// oscat_building/POUs/Jalousie/BLIND_CONTROL
FUNCTION_BLOCK BLIND_CONTROL
VAR_INPUT
	UP, DN : BOOL;
	S_IN : BYTE;
	PI : BYTE;
	AI : BYTE;
	T_UD, T_ANGLE : TIME;
END_VAR
VAR_INPUT CONSTANT
	SENS : BYTE := 5;
	T_LOCKOUT: TIME := T#100ms;
END_VAR
VAR_OUTPUT
	POS, ANG : BYTE;
	MU, MD : BOOL;
	STATUS : BYTE;
END_VAR
VAR
	act : BLIND_ACTUATOR;
	delta : BYTE;
	bTimeTest:BOOL:=FALSE;
	iPos:BYTE;
	iAngel:BYTE;
END_VAR

(*
version 1.5		8. mar 2011
programmer 		AE
tested by		AE

*)

IF bTimeTest THEN
	PI:=iPos;
	AI:=iAngel;
	UP:=TRUE;
	DN:=TRUE;
END_IF

(* Check Position*)
act(T_UD:=T_UD, T_ANGLE:=T_ANGLE, T_lockout := T_Lockout);

IF UP AND DN THEN
	(* automatic modus detected *)
	(* first find correct position *)
	IF BYTE_TO_INT(act.pos) < BYTE_TO_INT(pi) - delta THEN
		act.UP := TRUE;
		act.DN := FALSE;
		delta := 0;
		STATUS := 121;
	ELSIF BYTE_TO_INT(act.pos) > BYTE_TO_INT(pi) + delta THEN
		act.UP := FALSE;
		act.DN := TRUE;
		delta := 0;
		STATUS := 122;
	(* regulate angle *)
	ELSIF BYTE_TO_INT(act.ang) < BYTE_TO_INT(ai) - delta AND T_angle > T#100ms THEN
		act.UP := TRUE;
		act.DN := FALSE;
		delta := sens/2;
		STATUS := 123;
	ELSIF BYTE_TO_INT(act.ang) > BYTE_TO_INT(ai) + delta AND T_angle > T#100ms THEN
		act.UP := FALSE;
		act.DN := TRUE;
		delta := sens/2;
		STATUS := 124;
	(* correct position reached *)
	ELSE
		act.UP := FALSE;
		act.DN := FALSE;
		delta := sens;
		STATUS := S_IN;
	END_IF;
ELSE
	act.UP := UP;
	act.DN := DN;
	STATUS := S_IN;
END_IF;

(* blind control calls blind_actuator *)
act(T_UD:=T_UD, T_ANGLE:=T_ANGLE, T_lockout := T_Lockout);
pos := act.pos;
ang := act.ang;
MU := act.QU;
md := act.QD;
status := act.status;

(* revision history
hm	29. sep 2007	rev 1.0
	original release

hm	6. oct 2007	rev 1.1
	rearranged outputs
	integrated blind_actuator into blind_control

hm	16. oct 2007	rev 1.2
	ignore angle when t_angle = 0

hm 29. oct 2007	rev 1.3
	added lockout configuration time for motor direction change
	sens has a setup value of 5

hm	27. jul. 2009	rev 1.4
	changed status handling

ae	08. mar. 2010	rev 1.5
	at aPosition bevor control
	at tolerance "delta := sens/2;"

*)

END_FUNCTION_BLOCK

// oscat_building/POUs/Jalousie/BLIND_CONTROL_S
FUNCTION_BLOCK BLIND_CONTROL_S
VAR_INPUT
	UP, DN : BOOL;
	S_IN : BYTE := 125;
	PI : BYTE;
	T_UP : TIME;
	T_DN : TIME;
	RU : BOOL;
	RD : BOOL;
END_VAR
VAR_INPUT CONSTANT
	T_LOCKOUT: TIME := T#100ms;
	T_EXT : TIME;
	EXT_TRIG : BYTE := 5;
	R_POS_TOP : BYTE := 255;
	R_POS_BOT : BYTE;
END_VAR
VAR_OUTPUT
	POS : BYTE;
	MU, MD : BOOL;
	STATUS : BYTE;
END_VAR
VAR
	rmp : _RMP_NEXT;
	tx, last : TIME;
	PI_last: BYTE;
END_VAR


(*
version 1.2	23. jan 2010
programmer 	hugo
tested by		heinz


*)


(* status definition
	121 = manual up				manual up operation UP = true and DN = false
	122 = manual down			manual down operation DN = true and UP = false
	123 = auto positioning		automatic mode DN = UP = TRUE
	124 = revert					revert from top or bottom
	125 = nothing					default input for S_IN
	127 = Lockout time			lockout between directional change
	128 = calibrate				calibrate after power up
	129 = extend					extend runtime at top or bottom for continuous calibration
*)

(* read system time *)
tx := DWORD_TO_TIME(T_PLC_MS());

(* check inputs and start state machine *)
IF UP  AND NOT DN THEN
	(*  manual UP *)
	rmp.IN := 255;
	STATUS := 121;
ELSIF DN AND NOT UP THEN
	(* manual DN *)
	rmp.IN := 0;
	STATUS := 122;
ELSIF NOT (UP OR DN) THEN
	(* manual standby mode *)
	rmp.IN := PI;
	STATUS := S_IN;
END_IF;

(* simulate pos output *)
rmp(E := UP OR DN, TR := T_UP, TF := T_DN, TL := T_LOCKOUT, OUT := POS);

(* state machine *)
CASE STATUS OF
	0:		(* power up init *)
		last := tx;
		PI_last := PI XOR BYTE#255;
		STATUS := 128;		(* calibrate *)

	121: 	(* manual up *)
		MU := TRUE;
		MD := FALSE;
		IF POS >= (BYTE#255 - EXT_TRIG) THEN
			(* extend cycle if top is reached *)
			POS := 255;
			last := tx;
			STATUS := 129;	(* extend *)
		END_IF;

	122:	(* manual down *)
		MD := TRUE;
		MU := FALSE;
		IF POS <= EXT_TRIG THEN
			(* extend cycle if bottom is reached *)
			POS := 0;
			last := tx;
			STATUS := 129;	(* extend *)
		END_IF;

	123:	(* auto positioning *)
		MD := rmp.DN;
		MU := rmp.UP;
		IF NOT (rmp.DN OR rmp.UP) THEN
			(* automatic position is reached *)
			IF POS <= EXT_TRIG THEN
				(* extend at bottom *)
				MD := TRUE;
				last := tx;
				STATUS := 129;	(* extend *)
			ELSIF POS >= (BYTE#255 - EXT_TRIG)  THEN
				(* extend at top *)
				MU := TRUE;
				last := tx;
				STATUS := 129;	(* extend *)
			ELSE
				STATUS := S_IN;
			END_IF;
		END_IF;

	124:	(* revert from top or bottom *)
		MD := rmp.DN;
		MU := rmp.UP;
		IF NOT(rmp.DN OR rmp.UP) THEN
(*		IF POS = rmp.IN THEN  *)
			PI_last := PI;
			STATUS := S_IN;
		END_IF;

	127:	(* lockout time *)
		IF (tx - last) >= T_LOCKOUT THEN
				STATUS := S_IN;
		END_IF;

	128:	(* calibration *)
		MU := TRUE;
		MD := FALSE;
		rmp.IN := 255;
		IF (tx - last) >= (T_UP +  T_EXT) THEN
			MU := FALSE;
			last := tx;
			STATUS := 127;	(* lockout *)
		END_IF;

	129: (* extend mode *)
		IF (tx - last) >= T_EXT THEN
			MU := FALSE;
			MD := FALSE;
			last := tx;
			STATUS := 127;	(* lockout *)
		END_IF;

ELSE
	MU := FALSE;
	MD := FALSE;
	IF PI <> PI_last THEN
		PI_last := PI;
		rmp.IN := PI;
		STATUS := 123;	(* auto positioning *)
	ELSIF POS = 0 AND RU THEN
		rmp.IN := R_POS_BOT;
		STATUS := 124;	(* revert *)
	ELSIF pos = 255 AND RD THEN
		rmp.IN := R_POS_TOP;
		STATUS := 124;	(* revert *)
	ELSE
		STATUS := S_IN;
	END_IF;
END_CASE;



(* revision history

hm	9. mar. 2009	rev 1.0
	original release

hf	27. jul 2009	rev 1.1
	major code changes and updates

hf	23. Jan 2010	rev 1.2
	fixed a bug during calibration
	added T_UP and T_DN

*)

END_FUNCTION_BLOCK

// oscat_building/POUs/Jalousie/BLIND_INPUT
FUNCTION_BLOCK BLIND_INPUT
VAR_INPUT
	POS, ANG : BYTE;
	S1, S2 : BOOL;
	IN : BOOL;
	PI, AI : BYTE;
END_VAR
VAR_INPUT CONSTANT
	SINGLE_SWITCH : BOOL;
	CLICK_EN : BOOL := TRUE;
	CLICK_TIME : TIME := T#500ms;
	MAX_RUNTIME : TIME := T#60s;
	MANUAL_TIMEOUT: TIME := T#1h;
	DEBOUNCE_TIME : TIME := T#20ms;
	DBL_CLK1 : BOOL := FALSE;
	DBL_POS1 : BYTE;
	DBL_ANG1 : BYTE;
	DBL_CLK2 : BOOL := FALSE;
	DBL_POS2 : BYTE := 255;
	DBL_ANG2 : BYTE := 255;
	D1_TOGGLE : BOOL := TRUE;
	D2_TOGGLE : BOOL := TRUE;
	MASTER_MODE : BOOL;
END_VAR
VAR_OUTPUT
	QU : BOOL := TRUE;
	QD : BOOL := TRUE;
	STATUS : BYTE;
	PO : BYTE := 255;
	AO : BYTE := 255;
	D1, D2 : BOOL;
END_VAR
VAR
	s1e, s2e : TOF;
	s1d, s2d : CLICK_MODE;
	dir : BOOL;
	tx, last : TIME;
END_VAR

(*
version 1.7	12. nov. 2009
programmer 	hugo
tested by		oscat


*)

(* read system timer *)
tx := DWORD_TO_TIME(T_PLC_MS());

(* inputs S1 and S2 are debounced and then decoded for multiple clicks *)
s1e(in := S1, pt := DEBOUNCE_TIME);
s2e(in := S2, pt := DEBOUNCE_TIME);
s1d(in := (s1e.Q AND NOT SINGLE_SWITCH) OR (s1e.Q AND SINGLE_SWITCH AND dir), t_long := CLICK_TIME);
s2d(in := (s2e.Q AND NOT SINGLE_SWITCH) OR (s1e.Q AND SINGLE_SWITCH AND NOT dir), t_long := CLICK_TIME);

(* if d1 and d2 are not toggle clear them to make sure they are only active for oine cycle *)
IF NOT d1_toggle THEN d1 := FALSE; END_IF;
IF NOT d2_toggle THEN d2 := FALSE; END_IF;

(* decode actions *)
IF (s1d.LONG AND s2d.LONG) OR (status = 139) THEN
   status := 139;
   IF NOT (s1d.LONG OR s2d.LONG)  THEN status := 130; END_IF;
ELSIF s1d.tp_LONG THEN
	status := 132;
ELSIF s2d.tp_LONG THEN
	status := 133;
ELSIF  s1d.SINGLE THEN
	IF click_en THEN
		(* if running then we stop otherwise start new direction *)
		IF QU XOR QD THEN
			status := 131;
		ELSE
			status := 134;
			last := tx;
			dir := NOT dir;
		END_IF;
	END_IF;
ELSIF  s2d.SINGLE THEN
	IF click_en THEN
		(* if running then we stop otherwise start new direction *)
		IF QU XOR QD THEN
			status := 131;
		ELSE
			status := 135;
			last := tx;
			dir := NOT dir;
		END_IF;
	END_IF;
ELSIF in THEN
	status := 136;
	last := tx;
ELSIF s1d.DOUBLE THEN
	IF dbl_clk1 THEN
		(* a position need to be set for a double click on S1 *)
		status := 137;
		last := tx;
	ELSE
		(* toggle the output when dbl_clk1 is not active *)
		D1 := NOT D1;
	END_IF;
ELSIF s2d.DOUBLE THEN
	IF dbl_clk2 THEN
		(* a position need to be set for a double click on S2 *)
		status := 138;
		last := tx;
	ELSE
		(* toggle the output when dbl_clk2 is not active *)
		(* in single switch mode we need to toggle d1 instead of d2 *)
		IF single_switch THEN D1 := NOT D1; ELSE D2 := NOT D2; END_IF;
	END_IF;
END_IF;


(* state machine *)
CASE status OF
	0:		(* power up operation *)
			status := 130;

	130:	(* automatic operation standby *)
			IF NOT master_mode THEN
				PO := POS;
				AO := ANG;
			END_IF;
			QU := TRUE;
			QD := TRUE;

	131:	(* manual operation standby *)
			QU := FALSE;
			QD := FALSE;
			PO := POS;
			AO := ANG;
			(* manual mode will be ended when timeout is reached *)
			IF tx - last >= manual_timeout THEN
				status := 130;
			END_IF;

	132:	(* manual operation up *)
			QU := TRUE;
			QD := FALSE;
			PO := POS; AO := ANG;
			last := tx;
			IF NOT s1d.LONG THEN status := 131; dir := NOT dir; END_IF;

	133:	(* manual operation down *)
			QU := FALSE;
			QD := TRUE;
			PO := POS; AO := ANG;
			last := tx;
			IF NOT s2d.LONG THEN	status := 131; dir := NOT dir; END_IF;

	134:	(* manual operation single click up *)
			QU := TRUE;
			QD := FALSE;
			PO := POS; AO := ANG;
			IF tx - last >= max_runtime THEN status := 131; END_IF;

	135:	(* manual operation single click dn *)
			QU := FALSE;
			QD := TRUE;
			PO := POS; AO := ANG;
			IF tx - last >= max_runtime THEN status := 131;	END_IF;

	136:	(* forced input in = true *)
			QU := TRUE;
			QD := TRUE;
			PO := PI; AO := AI;
			IF tx-last >= max_runtime THEN status := 130; END_IF;

	137:	(* double click1 position *)
			QU := TRUE;
			QD := TRUE;
			PO := DBL_POS1;
			AO := DBL_ANG1;
			IF tx - last >= max_runtime THEN status := 131; END_IF;

	138:	(* double click2 position *)
			QU := TRUE;
			QD := TRUE;
			PO := DBL_POS2;
			AO := DBL_ANG2;
			IF tx - last >= max_runtime THEN status := 131; END_IF;

	   139:   (* manual operation standby *)
	         QU := FALSE;
	         QD := FALSE;
	         PO := POS;
	         AO := ANG;

END_CASE;


(* revision history
hm	29. sep 2007	rev 1.0
	original release

hm	6. oct 2007		rev 1.1
	renamed ps and as to po and ao

hm	30. dec 2007	rev 1.2
	added click_timeout variable and function

hm	16. jul. 2008	rev 1.3
	rewirtten code to allow for more functionality
	added single click mode with single_switch.
	added Debounce for inputs S1 and S2
	added double_click functionality

hm	26. sep. 2008	rev 1.4
	corrected an error while POS and ANG was transferred to outputs PO and AO during automatic modes

hm	22. jan 2009	rev 1.5
	added pulse mode for double click outputs
	added automatic mode for IN

hm	27. jul 2009	rev 1.6
	changed status 0 to 130

HF	12. nov. 2009	rev 1.7
	added state 139
	set defaults for QU, QD, PO

*)

END_FUNCTION_BLOCK

// oscat_building/POUs/Jalousie/BLIND_NIGHT
FUNCTION_BLOCK BLIND_NIGHT
VAR_INPUT
	UP, DN : BOOL;
	S_IN : BYTE;
	PI, AI : BYTE;
	E_NIGHT : BOOL := TRUE;
	E_DAY	: BOOL := TRUE;
	DTIN : DT;
	SUNRISE, SUNSET : TOD;
END_VAR
VAR_INPUT CONSTANT
	SUNRISE_OFFSET : TIME;
	SUNSET_OFFSET : TIME;
	NIGHT_POSITION : BYTE;
	NIGHT_ANGLE : BYTE;
END_VAR
VAR_OUTPUT
	QU, QD : BOOL;
	STATUS : BYTE;
	PO, AO : BYTE;
END_VAR
VAR
	night : BOOL;
	last_night, last_day : DATE;
END_VAR

(*
version 1.2	6 oct 2007
programmer 	hugo
tested by		tobias


*)

IF NOT (up AND dn) AND night THEN
	(* manual operation at night will cancel operation for one night *)
	night := FALSE;
ELSIF (DT_TO_TOD(dtin) > sunset + sunset_offset) AND (last_night < DT_TO_DATE(dtin)) AND NOT night AND e_night THEN
	(* enable night *)
	night := TRUE;
	last_night := DT_TO_DATE(dtin);
ELSIF (DT_TO_TOD(dtin) > sunrise + sunrise_offset) AND (last_day < DT_TO_DATE(dtin)) AND night AND e_day AND (last_night < DT_TO_DATE(dtin)) THEN
	(* disable night *)
	night := FALSE;
	last_day := DT_TO_DATE(dtin);
END_IF;

(* shade at night only in auto mode and enable = true *)
IF UP AND DN AND night THEN
	status := 141;
	po := night_position;
	ao := night_angle;
ELSE
	QU := UP;
	QD := DN;
	po := pi;
	ao := ai;
	status := s_in;
END_IF;


(* revision history
hm	29. sep 2007	rev 1.0
	original version

hm	5. oct 2007		rev 1.1
	added enable input

hm	6. oct 2007		rev 1.2
	added pos and angle inputs and outputs
	night position and angle can now be configured
	any manual operation at night will cancel night operation

*)

END_FUNCTION_BLOCK

// oscat_building/POUs/Jalousie/BLIND_SCENE
FUNCTION_BLOCK BLIND_SCENE
VAR_INPUT
	UP, DN : BOOL;
	S_IN : BYTE;
	PI, AI : BYTE;
	ENABLE : BOOL;
	SWRITE : BOOL;
	SCENE : BYTE;
END_VAR
VAR_OUTPUT
	QU, QD : BOOL;
	STATUS : BYTE;
	PO, AO : BYTE;
END_VAR
VAR RETAIN
	sx : ARRAY[0..15,0..2] OF BYTE;
END_VAR
VAR_TEMP
	x : BYTE;
END_VAR

(*
version 1.1	29. jan 2008
programmer 	hugo
tested by		tobias


*)

(* delete all bits except the lower 4 of scene *)
x := scene AND 16#0F;

IF enable AND sx[x,2] > 0 AND UP AND DN THEN
	po := sx[x,0];
	ao := sx[x,1];
	status := 160 + x;  (* Status number is 160 to 175 for the 16 scenes *)
	QU := TRUE;
	QD := TRUE;
ELSE
	QU := UP;
	QD := DN;
	status := S_IN;
	po := pi;
	ao := ai;
END_IF;

(* write scene if necessary *)
IF swrite THEN
	status := 176;		(* write scene *)
	sx[x,0] := pi;
	sx[x,1] := ai;
	IF enable THEN sx[x,2] := 1; ELSE sx[x,2] := 0; END_IF; (* if sx[x,2] = 0 the scene is disabled *)
END_IF;


(* revision history
hm	24. oct 2007	rev 1.0
	original release

hm		29.1.2008	rev 1.1
	replaced shr/shl with and for better performance
*)

END_FUNCTION_BLOCK

// oscat_building/POUs/Jalousie/BLIND_SECURITY
FUNCTION_BLOCK BLIND_SECURITY
VAR_INPUT
	UP, DN : BOOL;
	S_IN : BYTE;
	PI, AI : BYTE;
	FIRE : BOOL;
	WIND : BOOL;
	ALARM : BOOL;
	DOOR : BOOL;
	RAIN : BOOL;
END_VAR
VAR_INPUT CONSTANT
	Alarm_UP : BOOL := TRUE;
	WIND_UP :BOOL := TRUE;
	RAIN_UP : BOOL := FALSE;
END_VAR
VAR_OUTPUT
	QU, QD : BOOL;
	STATUS : BYTE;
	PO, AO : BYTE;
END_VAR


(*
version 1.2	12. feb 2008
programmer 	hugo
tested by		tobias


*)

IF Fire THEN
	QU := TRUE;
	QD := FALSE;
	status := 111;
ELSIF Wind THEN
	QU := Wind_up;
	QD := NOT wind_up;
	status := 112;
ELSIF alarm THEN
	QU := Alarm_up;
	QD := NOT Alarm_up;
	status := 113;
ELSIF Door THEN
	QU := TRUE;
	QD := FALSE;
	status := 114;
ELSIF Rain AND NOT (up XOR dn) THEN
	QU := rain_up;
	QD := NOT rain_up;
	status := 115;
ELSE
	QU := UP;
	QD := DN;
	status := S_IN;
	po := pi;
	ao := ai;
END_IF;


(* revision history
hm	29. sep 2007	rev 1.0
	original release

hm	6. oct 2007		rev 1.1
	added pos and angle inputs and outputs
	manual will override rain position
	alarm position can now be configured

hm		12. feb. 2008	rev 1.2
	added config variables rain_up and wind_up
	position for rain and wind is now configurable
*)

END_FUNCTION_BLOCK

// oscat_building/POUs/Jalousie/BLIND_SET
FUNCTION_BLOCK BLIND_SET
VAR_INPUT
	UP, DN : BOOL;
	S_IN : BYTE;
	PI, AI : BYTE;
	IN : BOOL;
	PX, AX : BYTE;
END_VAR
VAR_INPUT CONSTANT
	OVERRIDE_MANUAL : BOOL;
	RESTORE_POSITION : BOOL;
	RESTORE_TIME : TIME := T#60s;
END_VAR
VAR_OUTPUT
	QU, QD : BOOL;
	STATUS : BYTE;
	PO, AO : BYTE;
END_VAR
VAR
	tx: TIME;
	ps: BYTE;
	as: BYTE;
	last: TIME;
END_VAR

(*
version 1.0	27. jul 2009
programmer 	hugo
tested by		oscat

BLIND_SET can be used to force a definite position and angle.
blind_set can be placed close to blind_control for high priority while blind_input must be always at the beginning of the chain with low priority.

*)

(* read system time *)
tx := DWORD_TO_TIME(T_PLC_MS());

(* check inputs *)
IF IN THEN
	IF override_manual OR (UP AND DN) THEN
		status := 178;
	END_IF;
END_IF;

(* state machine *)
CASE STATUS OF
	0: (* power on state *)
		status := S_IN;

	178: (* force values from PX and AX *)
		PO := PX;
		AO := AX;
		QU := TRUE;
		QD := TRUE;
		(* check for end of forced position *)
		IF NOT in THEN
			STATUS := SEL(RESTORE_POSITION, S_IN, 179);
			last := tx;
		END_IF;

	179: (* restore previous position *)
		PO := ps;
		AO := as;
		IF ((PO = PI) AND (AO = AI))  OR tx - last >= RESTORE_TIME THEN
			status := S_IN;
		END_IF;

ELSE
	(* no operation transfer inputs to outputs *)
	PO := PI;
	ps := PI;
	AO := AI;
	as := AI;
	STATUS := S_IN;
	QU := UP;
	QD := DN;
END_CASE;


(* revision history
hm	27. jul 2009	rev 1.0
	original release

*)

END_FUNCTION_BLOCK

// oscat_building/POUs/Jalousie/BLIND_SHADE
FUNCTION_BLOCK BLIND_SHADE
VAR_INPUT
	UP, DN : BOOL;
	S_IN : BYTE;
	PI, AI : BYTE;
	ENABLE : BOOL;
	SUN : BOOL;
END_VAR
VAR_IN_OUT
	CX : CALENDAR;
END_VAR
VAR_INPUT CONSTANT
	sunrise_offset : TIME := T#1h;
	sunset_preset : TIME := T#1h;
	direction : REAL := 180.0;
	angle_offset : REAL := 80.0;
	slat_width : REAL := 80.0;
	Slat_spacing : REAL := 60.0;
	Shade_delay : TIME := T#60s;
	Shade_pos : BYTE;
END_VAR
VAR_OUTPUT
	QU, QD : BOOL;
	STATUS : BYTE;
	PO, AO : BYTE;
END_VAR
VAR
	angle: REAL;
	sun_delay : TOF;
END_VAR

(*
version 1.4	13. mar. 2009
programmer 	hugo
tested by		tobias


*)

(* the input sun is sent through tof which will delay the shade for the time shade_delay *)
sun_delay(IN := sun, PT := shade_delay);

IF UP AND DN AND enable AND sun_delay.Q AND cx.SUN_HOR > direction - angle_offset AND cx.SUN_HOR < direction + angle_offset AND
	DT_TO_TOD(cx.UTC) > cx.SUN_RISE + sunrise_offset AND DT_TO_TOD(cx.UTC) < cx.SUN_SET - sunset_preset THEN
	status := 151;
	QU := UP;
	QD := DN;
	(* position is predefined *)
	po := shade_pos;
	(* shading is active now calculate the slat angle *)
	(* calculate the max angle for the blind *)
	angle := DEG(ATAN(slat_spacing / slat_width));
	(* check if sun angle is between 0 and max angle *)
	IF cx.SUN_VER > 0.0 AND cx.SUN_VER < angle THEN
		angle := cx.SUN_VER + DEG(ACOS(COS(RAD(cx.SUN_VER))*slat_spacing / Slat_width));
		ao := DINT_TO_BYTE(LIMIT(0,TRUNC(angle * 2.833333333), 255));
	ELSE
		ao := 255;
	END_IF;
ELSE
	QU := UP;
	QD := DN;
	po := pi;
	ao := ai;
	status := S_IN;
END_IF;

(* revision history
hm	15 oct. 2007	rev 1.0
	original version

hm	19. oct 2007	rev 1.1
	manual mode was not detected because outputs were checked and not inputs UP and DN

hm	24. nov 2007	rev 1.2
	added shade_delay to avoid constant up and down if sun is out parcially

hm	8. feb 2009	rev 1.3
	added shading position shade_pos to be configured
	changed inputs to utilize calendar data structure

hm	13. mar. 2009	rev 1.4
	improved code

*)

END_FUNCTION_BLOCK

// oscat_building/POUs/Jalousie/BLIND_SHADE_S
FUNCTION_BLOCK BLIND_SHADE_S
VAR_INPUT
   UP, DN : BOOL;
   S_IN : BYTE;
   PI : BYTE;
   ENABLE : BOOL;
   SUN : BOOL;
   HORZ1 : REAL := 100.0;
   HORZ2 : REAL := 260.0;
   VERT : REAL := 90.0;
   ALERT: BOOL := FALSE;
END_VAR
VAR_IN_OUT
   CX : calendar;
END_VAR
VAR_INPUT CONSTANT
   sunrise_offset : TIME := T#1h;
   sunset_preset : TIME := T#1h;
   shade_delay : TIME := T#60s;
   shade_pos : BYTE;
END_VAR
VAR_OUTPUT
   QU, QD : BOOL;
   STATUS : BYTE;
   PO : BYTE;
END_VAR
VAR
   sun_delay : TOF;
END_VAR
(*
version 1.0	12. nov. 2009
programmer 	heinz
tested by		oscat


*)

(* status definition
   151 = shadow               move shutter down for shadowing
   152 = alert                  move shutter up by setting QU:=TRUE when door is open.
*)

(* the input sun is sent through tof which will delay the shade for the time shade_delay *)
sun_delay(IN := sun, PT := shade_delay);

IF ALERT THEN
   QU := TRUE;
   QD := FALSE;
   STATUS := 152;
ELSIF UP AND DN AND ENABLE AND sun_delay.Q
AND (CX.SUN_HOR > HORZ1) AND (CX.SUN_HOR < HORZ2)
AND (CX.SUN_VER < VERT)
AND (DT_TO_TOD(CX.UTC) > CX.SUN_RISE + sunrise_offset) AND (DT_TO_TOD(CX.UTC) < CX.SUN_SET - sunset_preset) THEN
   QU := UP;
   QD := DN;
   STATUS := 151;
   (* Calculate Position, must be shade_pos or less *)
   PO := MIN(PI, shade_pos);
ELSE
   QU := UP;
   QD := DN;
   PO := PI;
   STATUS := S_IN;
END_IF;



(* revision history
hf	12 nov. 2009	rev 1.0
	original version

*)

END_FUNCTION_BLOCK

// oscat_building/POUs/Other/BUILDING_VERSION
FUNCTION BUILDING_VERSION : DWORD
VAR_INPUT
	IN : BOOL;
END_VAR


(*
version 1.1	16 dec 2007
programmer 	hugo
tested by		oscat

oscat_version returns the version number in dword format
132 is library version 1.32
if IN = true, the release date will be returned

*)

IF in THEN
	BUILDING_VERSION := DATE_TO_DWORD(D#2011-02-3);
ELSE
	BUILDING_VERSION := 100;
END_IF;

(* revision history
hm	6. oct 2006	rev 1.0
	original version

hm	16. dec 2007	rev 1.1
	added possibility to return date and version depending on IN.

*)

END_FUNCTION

// oscat_network/POUs/CO_NVERT/BASE64_DECODE_STR_1
FUNCTION_BLOCK BASE64_DECODE_STR_1
VAR_INPUT
	RUN : BOOL;
END_VAR
VAR_OUTPUT
	DONE : BOOL;
END_VAR
VAR_IN_OUT
	STR1 : STRING(192);
	STR2 : STRING(144);
END_VAR
VAR
	BASE64_DECODE_STREAM : BASE64_DECODE_STREAM;
	run_last : BOOL;
	buf1 : ARRAY [0..63] OF BYTE;
	buf2 : ARRAY [0..47] OF BYTE;
	mode : INT;
	size1 : INT;
	size2 : INT;
	end : INT;
	pos : INT;
END_VAR

(*
version 1.0	06. dec. 2009
programmer 	ks
tested by	ks

BASE64_DECODE_STR konvertiert einen BASE64 kodierten String in einen normalen String. 

*)

CASE mode OF
0:	IF RUN AND NOT run_last THEN
		DONE := FALSE;
		mode := 1;
		end := LEN(STR1);
		pos := 0;
		STR2 := '';
	END_IF;
1:
	size1 := MIN(48,end - pos);
	IF size1 > 0 THEN
		_STRING_TO_BUFFER(STR:=MID(STR1, size1, pos + 1), POS:=0, PT:=ADR(buf1), SIZE:=SIZEOF(buf1));
		BASE64_DECODE_STREAM(BUF1:=buf1 ,BUF2:=buf2 ,SIZE1:=size1 ,SIZE2=>size2);
		STR2 := CONCAT(STR2,BUFFER_TO_STRING(PT:=ADR(buf2), SIZE:=SIZEOF(buf2), START:=0, STOP:=size2 - 1));
	ELSE
		mode := 0;
		DONE := TRUE;
	END_IF;
	pos := pos + size1;
END_CASE;

run_last := RUN;

(* revision history

ks	6. dec. 2009 rev 1.0
	original version

*)

END_FUNCTION_BLOCK

// oscat_network/POUs/CO_NVERT/BASE64_DECODE_STREAM_1
FUNCTION_BLOCK BASE64_DECODE_STREAM_1
VAR_IN_OUT
	BUF1 : ARRAY [0..63] OF BYTE;
	BUF2 : ARRAY [0..47] OF BYTE;
END_VAR
VAR_INPUT
	SIZE1 : INT;
END_VAR
VAR_OUTPUT
	SIZE2 : INT;
END_VAR
VAR_TEMP
	a: INT;
	b: WORD;
	o: INT;
	off: INT;
	i1: INT;
	i2: INT;
	c: INT;
END_VAR

(*
version 1.0	06. dec. 2009
programmer 	ks
tested by	ks

BASE64_DECODE_STREAM konvertiert einzelne Base64 kodierte Datenblöcke in normalen Datenblöcke. 

*)

IF SIZE1 <= 0 THEN SIZE2 := 0; RETURN; END_IF;
c := SIZE1 - 1;
i2 := 0;
a := 0;
b := 0;
FOR i1 := 0 TO c DO
	o := BUF1[i1];
	IF o = 61  (* = *) THEN	EXIT;
	ELSIF o > 96 (* a-z *) THEN off := 71;
	ELSIF o > 64 (* A-Z *) THEN off := 65;
	ELSIF o > 47 (* 0-9 *) THEN off := -4;
	ELSIF o = 43 (* + *) THEN off := -19;
	ELSIF o = 47 (* / *) THEN off := -16;
	END_IF;
	b := SHL(b,6) OR INT_TO_BYTE(o - off);
	a := a + 6;
	IF a >= 8 THEN
		a := a - 8;
		BUF2[i2] := WORD_TO_BYTE(SHR(b,a));
		i2 := i2 + 1;
		b := b AND NOT SHL(WORD#16#FFFF,a);
	END_IF;
END_FOR;
SIZE2 := i2;

(* revision history

ks	6. dec. 2009 rev 1.0
	original version

*)

END_FUNCTION_BLOCK

// oscat_network/POUs/CO_NVERT/BASE64_ENCODE_STR_1
FUNCTION_BLOCK BASE64_ENCODE_STR_1
VAR_INPUT
	RUN : BOOL;
END_VAR
VAR_OUTPUT
	DONE : BOOL;
END_VAR
VAR_IN_OUT
	STR1 : STRING(144);
	STR2 : STRING(192);
END_VAR
VAR
	BASE64_ENCODE_STREAM : BASE64_ENCODE_STREAM;
	run_last : BOOL;
	buf1 : ARRAY [0..47] OF BYTE;
	buf2 : ARRAY [0..63] OF BYTE;
	mode : INT;
	size1 : INT;
	size2 : INT;
	end : INT;
	pos : INT;
END_VAR

(*
version 1.0	06. dec. 2009
programmer 	ks
tested by	ks

BASE64_ENCODE_STR konvertiert einen normalen String in einen BASE64 kodierten String. 

*)

CASE mode OF
0:	IF RUN AND NOT run_last THEN
		DONE := FALSE;
		mode := 1;
		end := LEN(STR1);
		pos := 0;
		STR2 := '';
	END_IF;
1:
	size1 := MIN(48,end - pos);
	IF size1 > 0 THEN
		_STRING_TO_BUFFER(STR:=MID(STR1, size1, pos + 1), POS:=0, PT:=ADR(buf1), SIZE:=SIZEOF(buf1));
		BASE64_ENCODE_STREAM(BUF1:=buf1 ,BUF2:=buf2 ,SIZE1:=size1 ,SIZE2=>size2);
		STR2 := CONCAT(STR2,BUFFER_TO_STRING(PT:=ADR(buf2), SIZE:=SIZEOF(buf2), START:=0, STOP:=size2 - 1));
	ELSE
		mode := 0;
		DONE := TRUE;
	END_IF;
	pos := pos + size1;
END_CASE;

run_last := RUN;

(* revision history

ks	6. dec. 2009 rev 1.0
	original version

*)

END_FUNCTION_BLOCK

// oscat_network/POUs/CO_NVERT/BASE64_ENCODE_STREAM_1
FUNCTION_BLOCK BASE64_ENCODE_STREAM_1
VAR_IN_OUT
	BUF1 : ARRAY [0..47] OF BYTE;
	BUF2 : ARRAY [0..63] OF BYTE;
END_VAR
VAR_INPUT
	SIZE1 : INT;
END_VAR
VAR_OUTPUT
	SIZE2 : INT;
END_VAR
VAR
	a: INT;
	b: WORD;
	i: INT;
	i2: INT;
	i3: INT;
	c: INT;
	BASE64: STRING(64) := 'ABCDEFGHIJKLMNOPQRSTUVWXYZabcdefghijklmnopqrstuvwxyz0123456789+/';
END_VAR

(*
version 1.0	06. dec. 2009
programmer 	ks
tested by	ks

BASE64_ENCODE_STREAM konvertiert Datenblöcke in Base64. 

*)

IF SIZE1 <= 0 THEN
	SIZE2 := 0;
	RETURN;
END_IF;
c := SIZE1 - 1;
i2 := 0;
a := 0;
b := 0;
FOR i := 0 TO c DO
	b := SHL(b,8) OR BUF1[i];
	a := a + 8;
	WHILE a >= 6 DO
		a := a - 6;
		buf2[i2] := CODE(BASE64,WORD_TO_INT(SHR(b,a)) + 1);
		i2 := i2 + 1;
		b := b AND NOT SHL(WORD#16#FFFF,a);
	END_WHILE;
END_FOR;
IF a > 0 THEN
	buf2[i2] := CODE(BASE64,WORD_TO_INT(SHL(b,6 - a)) + 1);
	i2 := i2 + 1;
	i3 := i2 + (NOT INT_TO_WORD(i2) AND 2#11);
	FOR i := i2 TO i3 DO
		buf2[i] := 61;
	END_FOR;
	SIZE2 := i3 + 1;
ELSE
	SIZE2 := i2;
END_IF;

(* revision history

ks	6. dec. 2009 rev 1.0
	original version

*)

END_FUNCTION_BLOCK

// oscat_network/POUs/CO_NVERT/HTML_DECODE_1
FUNCTION HTML_DECODE_1 : STRING(STRING_LENGTH)
VAR_INPUT
	IN : STRING(STRING_LENGTH);
END_VAR
VAR
	pos : INT;
	end : INT;
	tmp : STRING(10);
	code : STRING(1);
END_VAR

(*
version 1.3		10. may 2010
programmer 	hugo
tested by		oscat

HTML_DECODE converts HTML coded characters to text. 
&amp; is replaced by & ("Ampersand")
&lt; is replaced by < ("lower than")
&gt; is replaced by > ("greater than")
&quot; is replaced by " ("Quote")
all other &names characters are replaced by their respective character codes.

*)

HTML_DECODE := IN;

(* docode characters encoded by character position *)
pos := FIND(HTML_DECODE, '&');
WHILE pos > 0 DO
	tmp := MID(HTML_DECODE, 2, pos + 1);
	IF tmp = '#x' OR tmp = '#X' THEN
		(* hexadecimal representation found *)
		tmp := MID(HTML_DECODE, 10, pos + 3);
		end := FIND(tmp, ';');
		CODE := CHR_TO_STRING(DWORD_TO_BYTE(HEX_TO_DWORD(LEFT(tmp, end - 1))));
		HTML_DECODE := REPLACE(HTML_DECODE, CODE, end + 3, pos);
	ELSIF LEFT(tmp,1) = '#' THEN
		tmp := MID(HTML_DECODE, 10, pos + 2);
		end := FIND(tmp, ';');
		CODE := CHR_TO_STRING(INT_TO_BYTE(STRING_TO_INT(LEFT(tmp, end - 1))));
		HTML_DECODE := REPLACE(HTML_DECODE, CODE, end + 2, pos);
	ELSE
		(* replace all named characters *)
		tmp := MID(HTML_DECODE, 10, pos + 1);
		end := FIND(tmp, ';');
		CODE := CHR_TO_STRING(CHARCODE(LEFT(tmp, end - 1)));
		HTML_DECODE := REPLACE(HTML_DECODE, CODE, end + 1, pos);
	END_IF;
	(* search for next occurence of encoded characters *)
	pos := FINDP(HTML_DECODE, '&', pos + 1);
END_WHILE;



(* revision history
hm	3. mai. 2008	rev 1.0
	original version

hm	16. jun. 2008	rev 1.1
	changed nested call of replace for better compatibility

hm	17. dec. 2008	rev 1.2
	changed function CHR to CHR_TO_STRING

hm	10. may. 2010	rev 1.3
	stringlength 250

*)

END_FUNCTION

// oscat_network/POUs/CO_NVERT/HTML_ENCODE_1
FUNCTION HTML_ENCODE_1 : STRING(STRING_LENGTH)
VAR_INPUT
	IN : STRING(STRING_LENGTH);
	M : BOOL;
END_VAR
VAR
	pt_in : POINTER TO ARRAY[1..255] OF BYTE;
	pt_out : POINTER TO ARRAY[1..256] OF BYTE;
	pos_in : INT;
	pos_out : INT;
	stop : INT;
	B: BYTE;
	tmp : STRING(10);
	i: INT;
END_VAR


(*
version 1.1		10. may. 2010
programmer 	hugo
tested by		hugo 

HTML_ENCODE checks a string if it contains reserved HTML characters and converts them to alternative html coding.
& is replaced by &amp; ("Ampersand")
< is replaced by &lt; ("lower than")
> is replaced by &gt; ("greater than")
" is replaced by &quot; ("Quote")

*)

pt_in  := ADR(in);
pt_out := ADR(HTML_ENCODE);

(* scan the input string and convert unallowed characters *)
pos_in := 1;
stop := LEN(in);
FOR pos_out := 1 TO 250 DO
	IF pos_in > stop THEN EXIT; END_IF;
	B := pt_in^[pos_in];
	CASE BYTE_TO_INT(B) OF
		34: (* " detected *)
			IF pos_out > STRING_LENGTH - 6 THEN EXIT; END_IF;
			pt_out^[pos_out] := 38;
			pos_out := pos_out + 1;
			pt_out^[pos_out] := 113;
			pos_out := pos_out + 1;
			pt_out^[pos_out] := 117;
			pos_out := pos_out + 1;
			pt_out^[pos_out] := 111;
			pos_out := pos_out + 1;
			pt_out^[pos_out] := 116;
			pos_out := pos_out + 1;
			pt_out^[pos_out] := 59;
		38: (* & detected *)
			IF pos_out > STRING_LENGTH - 5 THEN EXIT; END_IF;
			pt_out^[pos_out] := 38;
			pos_out := pos_out + 1;
			pt_out^[pos_out] := 97;
			pos_out := pos_out + 1;
			pt_out^[pos_out] := 109;
			pos_out := pos_out + 1;
			pt_out^[pos_out] := 112;
			pos_out := pos_out + 1;
			pt_out^[pos_out] := 59;
		60: (* < detected *)
			IF pos_out > STRING_LENGTH - 4 THEN EXIT; END_IF;
			pt_out^[pos_out] := 38;
			pos_out := pos_out + 1;
			pt_out^[pos_out] := 108;
			pos_out := pos_out + 1;
			pt_out^[pos_out] := 116;
			pos_out := pos_out + 1;
			pt_out^[pos_out] := 59;
		62: (* > detected *)
			IF pos_out > STRING_LENGTH - 4 THEN EXIT; END_IF;
			pt_out^[pos_out] := 38;
			pos_out := pos_out + 1;
			pt_out^[pos_out] := 103;
			pos_out := pos_out + 1;
			pt_out^[pos_out] := 116;
			pos_out := pos_out + 1;
			pt_out^[pos_out] := 59;
	ELSE
		IF M AND B > 127 THEN
			tmp := CHARNAME(B);
			(* exit if output string has not enough space *)
			IF pos_out + LEN(tmp) + 2 <= 250 THEN
				pt_out^[pos_out] := 38;
				pos_out := pos_out + 1;
				FOR i := 1 TO LEN(tmp) DO
					pt_out^[pos_out] := CODE(tmp, i);
					pos_out := pos_out + 1;
				END_FOR;
				pt_out^[pos_out] := 59;
			END_IF;
		ELSE
			pt_out^[pos_out] := B;
		END_IF;
	END_CASE;
	(* increment in by 1 *)
	pos_in := pos_in + 1;
END_FOR;

(* terminate the output string *)
pt_out^[pos_out] := 0;



(* revision history
hm		3. mai. 2008	rev 1.0
	original version

hm		10. mai. 2008	rev 1.1
	stringlength 250
*)

END_FUNCTION

// oscat_network/POUs/CO_NVERT/IP4_CHECK_1
FUNCTION IP4_CHECK_1 : BOOL
VAR_INPUT
	NIP : DWORD;
	LIP : DWORD;
	SM : DWORD;
END_VAR


(*
version 1.0	4. mar 2008
programmer 	hugo
tested by		oscat

IP4_CHECK testet ob eine Network IP und Local_IP im selben Subnet sind.

*)

IP4_CHECK := (NIP AND sm) = (LIP AND SM);


(* revision history
hm		4. mar 2008	rev 1.0
	original version

*)

END_FUNCTION

// oscat_network/POUs/CO_NVERT/IP4_DECODE_1
FUNCTION IP4_DECODE_1 : DWORD
VAR_INPUT
	str : STRING(15);
END_VAR
VAR
	pos: INT;
END_VAR

(*
version 1.1	10. mar 2009
programmer 	kurt
tested by		hugo

IP4_DECODE testet ob ein string eine gültige IPv4 Adresse enthält und gibt die 4 Bytes der IP Adresse als DWORD zurück.

*)

pos := FIND(str, '.');
WHILE pos > 0 DO
	IP4_DECODE := SHL(IP4_DECODE,8) OR STRING_TO_DWORD(LEFT(str,pos - 1));
	str := DELETE(str, pos, 1);
	pos := FIND(str, '.');
END_WHILE;
IP4_DECODE := SHL(IP4_DECODE,8) OR STRING_TO_DWORD(str);


(* revision history
hm		29. feb 2008	rev 1.0
	original version

hm	10. mar. 2009	rev 1.1
	new algorythm
*)

END_FUNCTION

// oscat_network/POUs/CO_NVERT/IP4_TO_STRING_1
FUNCTION IP4_TO_STRING_1 : STRING(15)
VAR_INPUT
	IP4 : DWORD;
END_VAR
VAR
	tmp : STRING(3);
END_VAR

(*
version 1.1	10. mar. 2009
programmer 	kurt
tested by	hugo

IP4_TO_STRING erzeugt eine IP Adresse als String aus einem DWORD..

*)

(* mask bits AND INSERT AT given position *)
tmp := BYTE_TO_STRING(DWORD_TO_BYTE(IP4));
IP4_TO_STRING := CONCAT('...', tmp);
tmp := BYTE_TO_STRING(DWORD_TO_BYTE(SHR(IP4,8)));
IP4_TO_STRING := INSERT(IP4_TO_STRING, tmp, 2);
tmp := BYTE_TO_STRING(DWORD_TO_BYTE(SHR(IP4,16)));
IP4_TO_STRING := INSERT(IP4_TO_STRING, tmp, 1);
tmp := BYTE_TO_STRING(DWORD_TO_BYTE(SHR(IP4,24)));
IP4_TO_STRING := CONCAT(tmp, IP4_TO_STRING);



(* revision history
hm	22. apr 2008	rev 1.0
	original version

hm	10. mar. 2009	rev 1.1
	improved code
*)

END_FUNCTION

// oscat_network/POUs/CO_NVERT/IS_IP4_1
FUNCTION IS_IP4_1 : BOOL
VAR_INPUT
	str : STRING;
END_VAR


(*
version 1.1	10. mar 2009
programmer 	kurt
tested by		hugo

IS_IP4 testet ob ein string eine gültige IPv4 Adresse enthält.

*)

IS_IP4 := COUNT_CHAR(str, 46) = 3;


(* revision history
hm	1. mar. 2008	rev 1.0
	original version

hm	10. mar. 2009	rev 1.1
	new code

*)

END_FUNCTION

// oscat_network/POUs/CO_NVERT/IS_URLCHR_1
FUNCTION IS_URLCHR_1 : BOOL
VAR_INPUT
	IN : BYTE;
END_VAR


(*
version 1.0		27. apr. 2008
programmer 		hugo
tested by		hugo

IS_URL_CHR is true if a string contains only non reserved characters for an url.
the non reserved characters are : [A..Z], [a..z], [0..9], -_.~

*)

IS_URLCHR := ((IN > 47) AND (IN < 58)) OR ((IN > 64) AND (IN < 91)) OR ((IN > 96) AND (IN < 123)) OR (in = 126) OR (in = 95) OR (in =45) OR (in =46);


(* revision history
hm		27. apr. 2008	rev 1.0
	original version

*)

END_FUNCTION

// oscat_network/POUs/CO_NVERT/MD5_AUX_1
FUNCTION MD5_AUX_1 : DWORD
VAR_INPUT
	N : INT;
	A : DWORD;
	B : DWORD;
	C : DWORD;
	D : DWORD;
	X : DWORD;
	U : INT;
	T : DWORD;
END_VAR
VAR
	w : DWORD;
END_VAR

(*
version 1.0	06. dec. 2009
programmer 	ks
tested by	ks

MD5_AUX ist ein Zusatzbaustein füR MD5_STREAM und enthäLT wiederkehrende Berechnungen
*)

CASE N OF
	1: w := (B AND C) OR (NOT(B) AND D);
	2: w := (B AND D) OR (C AND NOT D);
	3: w := (B XOR C XOR D);
	4: w := (C XOR (B OR  NOT(D)));
END_CASE

MD5_AUX := B + ROL(A + w + X + T,U);

(* revision history

ks	6. dec. 2009 rev 1.0
	original version

*)

END_FUNCTION

// oscat_network/POUs/CO_NVERT/MD5_CRAM_AUTH_1
FUNCTION_BLOCK MD5_CRAM_AUTH_1
VAR_IN_OUT
	RUN : BOOL;
	USERNAME : STRING(64);
	PASSWORD : STRING(64);
	B64_TS : STRING(64);  (* Base64 coded ServerTimeStamp *)
	AUTH_KEY : STRING(192);
END_VAR
VAR
	BASE64_DECODE_STR : BASE64_DECODE_STR;
	BASE64_ENCODE_STR : BASE64_ENCODE_STR;
	MD5_STREAM : MD5_STREAM;
	step : INT;
	md5_mode : INT;
	buf : ARRAY [0..63] OF BYTE;
	md5 : ARRAY [0..15] OF BYTE;
	md5_first : ARRAY [0..15] OF BYTE;
	md5_str1 : STRING(64);
	md5_str2 : STRING(64);
	size : UDINT;
	n1 : INT;
	n2 : INT;
	pos : UDINT;
	b64d_run : BOOL;
	b64d_done : BOOL;
	b64e_run : BOOL;
	b64e_done : BOOL;
	str_192 : STRING(192);
	str_144 : STRING(144);
	xpad : BYTE;
	pt : POINTER TO BYTE;
END_VAR

(*
version 1.0		10. may 2010
programmer 	ks
tested by		ks

Der Baustein MD5_CRAM_AUTH (Challenge-Response Authentication Mechanism, Message Digest 5) benutzt
das Authentifizierungsverfahren nach dem Challenge-Response-Prinzip auf der Basis des MD5-HMAC-Algorithmus.
Es wird beispielsweise zur Authentifizierung gegenüber SMTP- oder IMAP-Servern eingesetzt, da es die Übertragung des Passworts im Klartext vermeidet.
Durch dieses Verfahren kann auch über unverschlüsselte Kanäle eine sichere Authentifizierung gegenüber einem Server erfolgen


*)

CASE step OF

0:	IF RUN THEN
		step := 5;
		str_192 := B64_TS;
		b64d_run := TRUE;
	END_IF;

5: IF B64D_DONE THEN (* IPAD Zyklus *)
		b64d_run := FALSE;
		xpad := 16#36;
		md5_str1 := PASSWORD;
		md5_str2 := str_144;
		size := 64 + LEN(md5_str2);
		md5_mode := 1;
		step := 10;
	END_IF;

10: IF md5_mode = 3 THEN (* OPAD Zyklus *)
		md5_first := md5; (* md5 array vom IPAD sichern *)
		xpad := 16#5C;
		size := 64 + 16;
		md5_mode := 1;
		step := 20;
	END_IF;

20: IF md5_mode = 3 THEN
		md5_mode := 0;
		str_144 := CONCAT(USERNAME , ' ');
		str_144 := CONCAT(str_144 , MD5_TO_STRH(md5));
		b64e_run := TRUE;
		step := 30;
	END_IF;

30: IF B64E_DONE THEN
		AUTH_KEY := str_192;
		b64e_run := FALSE;
		RUN := FALSE;
		step := 0; (* alles beendet !! *)
	END_IF;

END_CASE;

(* ----------- md5 -------------- *)
CASE md5_mode OF

1:	n2 := LEN(md5_str1) - 1;
	pt := ADR(md5_str1);
	FOR n1 := 0 TO n2 DO (* string in buf kopieren *)
		buf[n1] := pt^ XOR xpad;
		pt := pt + 1;
	END_FOR;
	FOR n1 := n2 + 1 TO 63 DO (* mit ipad füllen *)
		buf[n1] := xpad;
	END_FOR;

2:	(* Data copy and Calc *)
	IF size > 0 AND pos >= 64 THEN
		IF step = 20 THEN
			FOR n1 := 0 TO 15 DO
				buf[n1] := md5_first[n1];
			END_FOR;
		ELSE
			n2 := LEN(md5_str2) - 1;
			pt := ADR(md5_str2);
			FOR n1 := 0 TO n2 DO (* string in buf kopieren *)
				buf[n1] := pt^;
				pt := pt + 1;
			END_FOR;
		END_IF;
	END_IF;

END_CASE;

IF md5_mode > 0 THEN
	MD5_STREAM(SIZE:=size, MODE:=md5_mode, BUF:=buf, MD5:=md5, POS=>pos);
END_IF;

BASE64_DECODE_STR(RUN:=b64d_run, STR1:=str_192, STR2:=str_144, DONE=>b64d_done);
BASE64_ENCODE_STR(RUN:=b64e_run, STR1:=str_144, STR2:=str_192, DONE=>b64e_done);

(* revision history

hm		10. mai. 2010	rev 1.0
	original version
*)

END_FUNCTION_BLOCK

// oscat_network/POUs/CO_NVERT/MD5_STR_1
FUNCTION_BLOCK MD5_STR_1
VAR_INPUT
	RUN: BOOL;
END_VAR
VAR_OUTPUT
	DONE: BOOL;
END_VAR
VAR_IN_OUT
	STR: STRING(STRING_LENGTH);
	MD5 : ARRAY [0..15] OF BYTE;
END_VAR
VAR
	run_last: BOOL;
	MD5_STREAM : MD5_STREAM;
	buf : ARRAY [0..63] OF BYTE;
	mode : INT;
	size : UDINT;
	pos : UDINT;
END_VAR

(*
version 1.0	06. dec. 2009
programmer 	ks
tested BY	ks

MD5_STR berechnet den MD5 Hash eines Strings
*)

CASE mode OF
0:	(* Wait für Start *)
	IF RUN AND NOT run_last THEN
		DONE := FALSE;
		mode := 1; (* Initialisierung *)
		size := LEN(STR);
	END_IF;

2:	(* Data copy and Calc *)
	IF size > 0 THEN
		_STRING_TO_BUFFER(STR:=MID(STR, UDINT_TO_INT(SIZE), UDINT_TO_INT(POS) + 1), POS:=0, PT:=ADR(buf), SIZE:=SIZEOF(buf));
	END_IF;

3:	DONE := TRUE;
	mode := 0; (* Stop *)

END_CASE;

IF mode > 0 THEN
	MD5_STREAM(SIZE:=size, MODE:=mode, BUF:=buf, MD5:=MD5, POS=>pos);
END_IF;

run_last := RUN;

(* revision history

ks	6. dec. 2009 rev 1.0
	original version

*)

END_FUNCTION_BLOCK

// oscat_network/POUs/CO_NVERT/MD5_STREAM_1
FUNCTION_BLOCK MD5_STREAM_1
VAR_IN_OUT
	MODE : INT;
	BUF : ARRAY [0..63] OF BYTE;
	MD5 : ARRAY [0..15] OF BYTE;
	SIZE : UDINT;
END_VAR

VAR_OUTPUT
	POS : UDINT;
END_VAR

VAR
	hash : ARRAY [0..3] OF DWORD;
	a : DWORD;
	b : DWORD;
	c : DWORD;
	d : DWORD;
	end : UDINT;
	block : UDINT;
	x : ARRAY [0..15] OF DWORD;
	n : INT;
	n1 : INT;
	z : INT;
	pad_1 : BOOL;
END_VAR

(*
version 1.0	06. dec. 2009
programmer 	ks
tested BY	ks

MD5_STREAM berechnet den MD5 Hash eines Datenstromes
*)

CASE MODE OF

1:	(* Initialisierung der Hash-Werte *)
	hash[0] := DWORD#16#67452301;
	hash[1] := DWORD#16#EFCDAB89;
	hash[2] := DWORD#16#98BADCFE;
	hash[3] := DWORD#16#10325476;

	block := SHR(SIZE,6) + BOOL_TO_UDINT((UDINT_TO_BYTE(SIZE) AND 16#3F) > 55);
	pad_1 := FALSE;
	POS := 0;
	End := SIZE;
	SIZE := MIN(64,End);
	MODE := 2;

2:	(* Fuell-Bytes anhängen *)
	FOR n := UDINT_TO_INT(SIZE) TO 63 DO
		BUF[n] := 0;
	END_FOR;

	IF SIZE < 64 AND NOT pad_1 THEN
		BUF[SIZE] := 2#1000_0000;
		pad_1 := TRUE;
	END_IF;

	POS := POS + SIZE;
	SIZE := MIN(64,End - POS);

	n := 0;	(* Byte-Array in DWORD-Array umkopieren *)
	FOR n1 := 0 TO 15 DO
		x[n1] := DWORD_OF_BYTE(BUF[n+3],BUF[n+2],BUF[n+1],BUF[n]); (* Little Endian Format *)
		n := n + 4;
	END_FOR;

	IF block = 0 THEN (* am Ende des letzten Blocks die Datenlänge eintragen *)
		x[14] := SHL(UDINT_TO_DWORD(End),3); (* Anzahl Datenbits im Little-Endian Format eintragen *)
		MODE := 3;
	ELSE
		block := block - 1;
	END_IF;

	a := hash[0];
	b := hash[1];
	c := hash[2];
	d := hash[3];

	a := MD5_AUX(1, a, b, c, d, X[00], 07, 16#D76AA478); (* 01 *)
	d := MD5_AUX(1, d, a, b, c, X[01], 12, 16#E8C7B756); (* 02 *)
	c := MD5_AUX(1, c, d, a, b, X[02], 17, 16#242070DB); (* 03 *)
	b := MD5_AUX(1, b, c, d, a, X[03], 22, 16#C1BDCEEE); (* 04 *)
	a := MD5_AUX(1, a, b, c, d, X[04], 07, 16#F57C0FAF); (* 05 *)
	d := MD5_AUX(1, d, a, b, c, X[05], 12, 16#4787C62A); (* 06 *)
	c := MD5_AUX(1, c, d, a, b, X[06], 17, 16#A8304613); (* 07 *)
	b := MD5_AUX(1, b, c, d, a, X[07], 22, 16#FD469501); (* 08 *)
	a := MD5_AUX(1, a, b, c, d, X[08], 07, 16#698098D8); (* 09 *)
	d := MD5_AUX(1, d, a, b, c, X[09], 12, 16#8B44F7AF); (* 10 *)
	c := MD5_AUX(1, c, d, a, b, X[10], 17, 16#FFFF5BB1); (* 11 *)
	b := MD5_AUX(1, b, c, d, a, X[11], 22, 16#895CD7BE); (* 12 *)
	a := MD5_AUX(1, a, b, c, d, X[12], 07, 16#6B901122); (* 13 *)
	d := MD5_AUX(1, d, a, b, c, X[13], 12, 16#FD987193); (* 14 *)
	c := MD5_AUX(1, c, d, a, b, X[14], 17, 16#A679438E); (* 15 *)
	b := MD5_AUX(1, b, c, d, a, X[15], 22, 16#49B40821); (* 16 *)

	a := MD5_AUX(2, a, b, c, d, X[01], 05, 16#F61E2562); (* 17 *)
	d := MD5_AUX(2, d, a, b, c, X[06], 09, 16#C040B340); (* 18 *)
	c := MD5_AUX(2, c, d, a, b, X[11], 14, 16#265E5A51); (* 19 *)
	b := MD5_AUX(2, b, c, d, a, X[00], 20, 16#E9B6C7AA); (* 20 *)
	a := MD5_AUX(2, a, b, c, d, X[05], 05, 16#D62F105D); (* 21 *)
	d := MD5_AUX(2, d, a, b, c, X[10], 09, 16#02441453); (* 22 *)
	c := MD5_AUX(2, c, d, a, b, X[15], 14, 16#D8A1E681); (* 23 *)
	b := MD5_AUX(2, b, c, d, a, X[04], 20, 16#E7D3FBC8); (* 24 *)
	a := MD5_AUX(2, a, b, c, d, X[09], 05, 16#21E1CDE6); (* 25 *)
	d := MD5_AUX(2, d, a, b, c, X[14], 09, 16#C33707D6); (* 26 *)
	c := MD5_AUX(2, c, d, a, b, X[03], 14, 16#F4D50D87); (* 27 *)
	b := MD5_AUX(2, b, c, d, a, X[08], 20, 16#455A14ED); (* 28 *)
	a := MD5_AUX(2, a, b, c, d, X[13], 05, 16#A9E3E905); (* 29 *)
	d := MD5_AUX(2, d, a, b, c, X[02], 09, 16#FCEFA3F8); (* 30 *)
	c := MD5_AUX(2, c, d, a, b, X[07], 14, 16#676F02D9); (* 31 *)
	b := MD5_AUX(2, b, c, d, a, X[12], 20, 16#8D2A4C8A); (* 32 *)

	a := MD5_AUX(3, a, b, c, d, X[05], 04, 16#FFFA3942); (* 33 *)
	d := MD5_AUX(3, d, a, b, c, X[08], 11, 16#8771F681); (* 34 *)
	c := MD5_AUX(3, c, d, a, b, X[11], 16, 16#6D9D6122); (* 35 *)
	b := MD5_AUX(3, b, c, d, a, X[14], 23, 16#FDE5380C); (* 36 *)
	a := MD5_AUX(3, a, b, c, d, X[01], 04, 16#A4BEEA44); (* 37 *)
	d := MD5_AUX(3, d, a, b, c, X[04], 11, 16#4BDECFA9); (* 38 *)
	c := MD5_AUX(3, c, d, a, b, X[07], 16, 16#F6BB4B60); (* 39 *)
	b := MD5_AUX(3, b, c, d, a, X[10], 23, 16#BEBFBC70); (* 40 *)
	a := MD5_AUX(3, a, b, c, d, X[13], 04, 16#289B7EC6); (* 41 *)
	d := MD5_AUX(3, d, a, b, c, X[00], 11, 16#EAA127FA); (* 42 *)
	c := MD5_AUX(3, c, d, a, b, X[03], 16, 16#D4EF3085); (* 43 *)
	b := MD5_AUX(3, b, c, d, a, X[06], 23, 16#04881D05); (* 44 *)
	a := MD5_AUX(3, a, b, c, d, X[09], 04, 16#D9D4D039); (* 45 *)
	d := MD5_AUX(3, d, a, b, c, X[12], 11, 16#E6DB99E5); (* 46 *)
	c := MD5_AUX(3, c, d, a, b, X[15], 16, 16#1FA27CF8); (* 47 *)
	b := MD5_AUX(3, b, c, d, a, X[02], 23, 16#C4AC5665); (* 48 *)

	a := MD5_AUX(4, a, b, c, d, X[00], 06, 16#F4292244); (* 49 *)
	d := MD5_AUX(4, d, a, b, c, X[07], 10, 16#432AFF97); (* 50 *)
	c := MD5_AUX(4, c, d, a, b, X[14], 15, 16#AB9423A7); (* 51 *)
	b := MD5_AUX(4, b, c, d, a, X[05], 21, 16#FC93A039); (* 52 *)
	a := MD5_AUX(4, a, b, c, d, X[12], 06, 16#655B59C3); (* 53 *)
	d := MD5_AUX(4, d, a, b, c, X[03], 10, 16#8F0CCC92); (* 54 *)
	c := MD5_AUX(4, c, d, a, b, X[10], 15, 16#FFEFF47D); (* 55 *)
	b := MD5_AUX(4, b, c, d, a, X[01], 21, 16#85845DD1); (* 56 *)
	a := MD5_AUX(4, a, b, c, d, X[08], 06, 16#6FA87E4F); (* 57 *)
	d := MD5_AUX(4, d, a, b, c, X[15], 10, 16#FE2CE6E0); (* 58 *)
	c := MD5_AUX(4, c, d, a, b, X[06], 15, 16#A3014314); (* 59 *)
	b := MD5_AUX(4, b, c, d, a, X[13], 21, 16#4E0811A1); (* 60 *)
	a := MD5_AUX(4, a, b, c, d, X[04], 06, 16#F7537E82); (* 61 *)
	d := MD5_AUX(4, d, a, b, c, X[11], 10, 16#BD3AF235); (* 62 *)
	c := MD5_AUX(4, c, d, a, b, X[02], 15, 16#2AD7D2BB); (* 63 *)
	b := MD5_AUX(4, b, c, d, a, X[09], 21, 16#EB86D391); (* 64 *)

	hash[0] := hash[0] + a;
	hash[1] := hash[1] + b;
	hash[2] := hash[2] + c;
	hash[3] := hash[3] + d;

END_CASE;

IF MODE = 3 THEN
	z := 0;
	FOR n := 0 TO 3 DO (* von Little-Endian auf Big-Endian format konvertieren und DWORD auf BYTE-Array *)
		FOR n1 := 0 TO 3 DO
			MD5[z] := DWORD_TO_BYTE(hash[n]);
			hash[n] := ROR(hash[n],8);
			z := z + 1;
		END_FOR;
	END_FOR;
END_IF;

(* revision history

ks	6. dec. 2009 rev 1.0
	original version

*)

END_FUNCTION_BLOCK

// oscat_network/POUs/CO_NVERT/MD5_TO_STRH_1
FUNCTION MD5_TO_STRH_1 : STRING(32)
VAR_INPUT
	MD5 : ARRAY [0..15] OF BYTE;
END_VAR
VAR
	i : INT;
	tmp : BYTE;
	pt : POINTER TO BYTE;
END_VAR
(*
version 1.0	06. dec. 2009
programmer 	ks
tested BY	ks

MD5_TO_STRH konvertiert das MD5 Hash Array in einen HEX-String
*)

pt := ADR(MD5_TO_STRH); (* read output adress to pointer *)

FOR i := 0 TO 15 DO; (* write the 8 hex characters backwards *)
	tmp := SHR(MD5[i],4);
	PT^ := tmp + SEL(tmp <= 9,87,48);
	pt := pt + 1; (* decrement the pointer *)
	tmp := MD5[i] AND 2#1111;
	PT^ := tmp + SEL(tmp <= 9,87,48);
	pt := pt + 1; (* decrement the pointer *)
END_FOR;
pt^:= 0; (* write the closing byte for the string *)

(* revision history

ks	6. dec. 2009 rev 1.0
	original version

*)

END_FUNCTION

// oscat_network/POUs/CO_NVERT/RC4_CRYPT_STREAM_1
FUNCTION_BLOCK RC4_CRYPT_STREAM_1
VAR_IN_OUT
	MODE : INT;
	KEY : STRING(40);
	BUF : ARRAY [0..63] OF BYTE;
	SIZE : UDINT;
END_VAR

VAR_OUTPUT
	POS : UDINT;
END_VAR

VAR
	sbox : ARRAY [0..255] OF BYTE;
	skey : ARRAY [0..255] OF BYTE;
	a : INT;
	b : INT;
	c : INT;
	d : USINT;
	e : USINT;
	end : UDINT;
	v : BYTE;
END_VAR

(*
version 1.0	09. jan. 2010
programmer	ks
tested BY	ks

RC4_CRYPT_STREAM kann einen Datenstrom ver/entschlüsseln mittels der RC4 Stromchiffrierung
*)

CASE MODE OF

1:	(* Initialisierung *)
	b := LEN(KEY) - 1;
	IF b < 0 OR SIZE < 1 THEN
		MODE := 3;
		RETURN;
	END_IF;

	FOR a := 0 TO b DO
		skey[a] := CODE(KEY, a + 1);
		sbox[a] := INT_TO_BYTE(a);
	END_FOR;

	c := 0;
	FOR a := b + 1 TO 255 DO
		skey[a] := skey[c];
		sbox[a] := INT_TO_BYTE(a);
		c := c + 1;
		IF c > b THEN c := 0; END_IF;
	END_FOR;

	d := 0;
	FOR a := 0 TO 255 DO
		d := d + sbox[a] + skey[a];
		v := sbox[a];
		sbox[a] := sbox[d];
		sbox[d] := v;
	END_FOR;

	POS := 0;
	end := SIZE;
	SIZE := MIN(64,end);
	d := 0;
	e := 0;
	MODE := 2;

2:	(* Daten ver/entschlüsseln *)

	b := UDINT_TO_INT(SIZE) - 1;
	FOR a := 0 TO b DO
		d := d + 1;
		e := e + sbox[d];
		v := sbox[d];
		sbox[d] := sbox[e];
		sbox[e] := v;
		v := sbox[d] + sbox[e];
		BUF[a] :=BUF[a] XOR sbox[v];
	END_FOR;

	POS := POS + SIZE;
	SIZE := MIN(64,end - POS);

	IF SIZE = 0 THEN
		MODE := 3;
	END_IF;
END_CASE;

(* revision history

ks	9. Jan. 2010 rev 1.0
	original version

*)

END_FUNCTION_BLOCK

// oscat_network/POUs/CO_NVERT/SHA1_STR_1
FUNCTION_BLOCK SHA1_STR_1
VAR_INPUT
	RUN: BOOL;
END_VAR
VAR_OUTPUT
	DONE: BOOL;
END_VAR
VAR_IN_OUT
	STR: STRING(STRING_LENGTH);
	SHA1 : ARRAY [0..19] OF BYTE;
END_VAR

VAR
	run_last: BOOL;
	SHA1_STREAM : SHA1_STREAM;
	buf : ARRAY [0..63] OF BYTE;
	mode : INT;
	size : UDINT;
	pos : UDINT;
END_VAR

(*
version 1.0	06. dec. 2009
programmer 	ks
tested BY	ks

SHA1_STR berechnet den MD5 Hash eines Strings
*)

CASE mode OF
0:	(* Wait für Start *)
	IF RUN AND NOT run_last THEN
		DONE := FALSE;
		mode := 1; (* Initialisierung *)
		size := LEN(STR);
	END_IF;

2:	(* Data copy and Calc *)
	IF size > 0 THEN
		_STRING_TO_BUFFER(STR:=MID(STR, UDINT_TO_INT(SIZE), UDINT_TO_INT(POS) + 1), POS:=0, PT:=ADR(buf), SIZE:=SIZEOF(buf));
	END_IF;

3:	DONE := TRUE;
	mode := 0; (* Stop *)

END_CASE;

IF mode > 0 THEN
	SHA1_STREAM(SIZE:=size, MODE:=mode, BUF:=buf, SHA1:=SHA1, POS=>pos);
END_IF;

run_last := RUN;

(* revision history

ks	6. dec. 2009 rev 1.0
	original version

*)

END_FUNCTION_BLOCK

// oscat_network/POUs/CO_NVERT/SHA1_STREAM_1
FUNCTION_BLOCK SHA1_STREAM_1
VAR_IN_OUT
	MODE : INT;
	BUF : ARRAY [0..63] OF BYTE;
	SHA1 : ARRAY [0..19] OF BYTE;
	SIZE : UDINT;
END_VAR

VAR_OUTPUT
	POS : UDINT;
END_VAR

VAR
	hash : ARRAY [0..4] OF DWORD;
	end : UDINT;
	block : UDINT;
	pad_1 : BOOL;
	w : ARRAY [0..79] OF DWORD;
	n : INT;
	n1 : INT;
	a : DWORD;
	b : DWORD;
	c : DWORD;
	d : DWORD;
	e : DWORD;
	f : DWORD;
	k : DWORD;
	x : DWORD;
	z : INT;
END_VAR

(*
version 1.0	06. dec. 2009
programmer 	ks
tested BY	ks

SHA1_STREAM berechnet den SHA1 Hash eines Datenstromes
*)

CASE MODE OF

1:	(* Initialisierung der Hash-Werte *)
	hash[0] := DWORD#16#67452301;
	hash[1] := DWORD#16#EFCDAB89;
	hash[2] := DWORD#16#98BADCFE;
	hash[3] := DWORD#16#10325476;
	hash[4] := DWORD#16#C3D2E1F0;

	(* Buffer initialisieren *)
	FOR n := 16 TO 79 DO
   		w[n] := DWORD#0;
	END_FOR;

	block := SHR(SIZE,6) + BOOL_TO_UDINT((UDINT_TO_BYTE(SIZE) AND 16#3F) > 55);	(* benötigte Blocks errechnen *)

	pad_1 := FALSE;
	POS := 0;
	End := SIZE;
	SIZE := MIN(64,End);
	MODE := 2;

2:	FOR n := UDINT_TO_INT(SIZE) TO 63 DO (* Fuell-Bytes anhängen *)
		BUF[n] := 0;
	END_FOR;

	IF SIZE < 64 AND NOT pad_1 THEN
		BUF[SIZE] := 2#1000_0000;
		pad_1 := TRUE;
	END_IF;

	POS := POS + SIZE;
	SIZE := MIN(64,End - POS);

	n := 0;	(* Byte-Array in DWORD-Array umkopieren *)
	FOR n1 := 0 TO 15 DO
		w[n1] := DWORD_OF_BYTE(BUF[n],BUF[n+1],BUF[n+2],BUF[n+3]);
		n := n + 4;
	END_FOR;

	IF block = 0 THEN (* am Ende des letzten Blocks die Datenlänge eintragen *)
		w[15] := SHL(UDINT_TO_DWORD(End),3); (* Anzahl Datenbits eintragen *)
		MODE := 3;
	ELSE
		block := block - 1;
	END_IF;

	FOR n := 16 TO 79 DO (* erweitern der 16 32-bit-Worte auf 80 32-bit-Worte *)
		w[n] := ROL(w[n-3] XOR w[n-8] XOR w[n-14] XOR w[n-16],1);
	END_FOR;

	a := hash[0];
	b := hash[1];
	c := hash[2];
	d := hash[3];
	e := hash[4];

	FOR n := 0 TO 79 DO
		IF n <= 19 THEN
			f := (b AND c) OR (NOT(b) AND d);
			k := DWORD#16#5A827999;
		ELSIF n <= 39 THEN
			f := b XOR c XOR d;
			k := DWORD#16#6ED9EBA1;
		ELSIF n <= 59 THEN
			f := (b AND c) OR (b AND d) OR (c AND d);
			k := DWORD#16#8F1BBCDC;
		ELSE
			f := b XOR c XOR d;
			k := DWORD#16#CA62C1D6;
		END_IF;

		x := ROL(a,5) + f + e + k + w[n];
		e := d;
		d := c;
		c := ROL(b,30);
		b := a;
		a := x;
	END_FOR;

	(* aktuelle Hash-Werte zum letzten Wert addieren *)
	hash[0] := hash[0] + a;
	hash[1] := hash[1] + b;
	hash[2] := hash[2] + c;
	hash[3] := hash[3] + d;
	hash[4] := hash[4] + e;

END_CASE;

IF MODE = 3 THEN
	z := 0;
	FOR n := 0 TO 4 DO (* konvertiere DWORD auf BYTE-Array *)
		FOR n1 := 0 TO 3 DO
			hash[n] := ROL(hash[n],8);
			SHA1[z] := DWORD_TO_BYTE(hash[n]);
			z := z + 1;
		END_FOR;
	END_FOR;
END_IF;

(* revision history

ks	6. dec. 2009 rev 1.0
	original version

*)

END_FUNCTION_BLOCK

// oscat_network/POUs/CO_NVERT/SHA1_TO_STRH_1
FUNCTION SHA1_TO_STRH_1 : STRING(40)
VAR_INPUT
	SHA1 : ARRAY [0..19] OF BYTE;
END_VAR
VAR
	i : INT;
	tmp : BYTE;
	pt : POINTER TO BYTE;
END_VAR
(*
version 1.1	03. dec. 2011
programmer 	ks
tested BY	ks

SHA1_TO_STRH konvertiert das SHA1 Hash Array in einen HEX-String
*)

pt := ADR(SHA1_TO_STRH); (* read output adress to pointer *)

FOR i := 0 TO 19 DO; (* write the 10 hex characters backwards *)
	tmp := SHR(SHA1[i],4);
	PT^ := tmp + SEL(tmp <= 9,87,48);
	pt := pt + 1; (* decrement the pointer *)
	tmp := SHA1[i] AND 2#1111;
	PT^ := tmp + SEL(tmp <= 9,87,48);
	pt := pt + 1; (* decrement the pointer *)
END_FOR;
pt^:= 0; (* write the closing byte for the string *)

(* revision history

ks	6. dec. 2009 rev 1.0
	original version

ks	3. dec. 2011 rev 1.1
	incorrect string size
*)

END_FUNCTION

// oscat_network/POUs/CO_NVERT/STRING_TO_URL_1
FUNCTION STRING_TO_URL_1 : URL
VAR_INPUT
	STR : STRING(STRING_LENGTH);
	DEFAULT_PROTOCOL : STRING(10);
	DEFAULT_PATH : STRING(80);
END_VAR
VAR
	pos: INT;
	pos2: INT;
END_VAR
VAR_TEMP
	x : STRING(STRING_LENGTH);
END_VAR

(*
version 1.1	20. dec. 2010
programmer 	hugo
tested by		oscat

URL splits a unifrom resource locator in its conponents.

*)

(*

http://hans:geheim@www.example.org:80/demo/example.cgi?land=de&stadt=aa#abschnitt1
|       |      |         |         |   |                   |               |
|       |      |         Host      |   Pfad                Query           Anker
|       |      Passwort            Port
|       Benutzer
Protokoll

*)

(* check if string is empty and return empty url *)
IF STR = '' THEN RETURN; END_IF;

(* extract the protocol *)
(* first we check if the optional protocol is specified ending with a :// *)
pos := FIND(STR, '://');
IF pos > 0 THEN
	(* store protocol and restore the rest of url in temp *)
	STRING_TO_URL.PROTOCOL := LEFT(STR, pos - 1);
	x := RIGHT(STR, LEN(STR) - pos - 2);
ELSE
	x := STR;
	STRING_TO_URL.PROTOCOL := DEFAULT_PROTOCOL;
END_IF;

(* extract user and password if present ending with a @ *)
pos := FIND(x, '@');
IF pos > 0 THEN
	(* extract user *)
	pos2 := FIND(x,':')+1;
	IF pos2 > 1 AND pos2 <= pos THEN
		STRING_TO_URL.USER := LEFT(x,pos2 - 2);
		STRING_TO_URL.PASSWORD := MID(x, pos - pos2, pos2);
	ELSE
		STRING_TO_URL.USER := LEFT(x, pos - 2);
		STRING_TO_URL.PASSWORD := '';
	END_IF;
	x := RIGHT(x, LEN(x) - pos);
ELSE
	STRING_TO_URL.USER := '';
	STRING_TO_URL.PASSWORD := '';
END_IF;

(* extract anchor *)
pos := FIND(x, '#');
IF pos > 0 THEN
	STRING_TO_URL.ANCHOR := RIGHT(x, LEN(x) - pos);
	x := LEFT(x, pos - 1);
ELSE
	STRING_TO_URL.ANCHOR := '';
END_IF;

(* extract query  *)
pos := FIND(x, '?');
IF pos > 0 THEN
	STRING_TO_URL.QUERY := RIGHT(x, LEN(x) - pos);
	x := LEFT(x, pos - 1);
ELSE
	STRING_TO_URL.QUERY := '';
END_IF;

(* extract path  *)
pos := FIND(x, '/');
IF pos > 0 THEN
	STRING_TO_URL.PATH := RIGHT(x, LEN(x) - pos + 1);
	x := LEFT(x, pos - 1);
ELSE
	STRING_TO_URL.PATH := DEFAULT_PATH;
END_IF;

(* extract port and leave domain *)
pos := FIND(x, ':');
IF pos > 0 THEN
	STRING_TO_URL.PORT := STRING_TO_WORD(RIGHT(x, LEN(x) - pos));
	STRING_TO_URL.DOMAIN := LEFT(x, pos - 1);
ELSE
	STRING_TO_URL.PORT := 0;
	STRING_TO_URL.DOMAIN := x;
END_IF;

(* revision history
hm		18. apr 2008	rev 1.0
	original version

ks		20. dec. 2010	rev 1.1
	stringlength 250 , var x

*)

END_FUNCTION

// oscat_network/POUs/CO_NVERT/URL_DECODE_1
FUNCTION URL_DECODE_1 : STRING(STRING_LENGTH)
VAR_INPUT
	IN : STRING(STRING_LENGTH);
END_VAR
VAR
	pos : INT;
	seq : STRING(3);
	new : STRING(1);
END_VAR


(*
version 1.2		10. may. 2010
programmer 	hugo
tested by		hugo

URL_DECODE checks a string if it contains non reserved characters represented by a % followed with the two digit hex code and converts them to their ascii code.
the non reserved characters are : [A..Z], [a..z], [0..9], -_.~
for example the character sequence '%23' will be converted to '#'.

*)

URL_DECODE := IN;
pos := FIND(URL_DECODE,'%');
WHILE pos > 0 DO
	seq := MID(URL_DECODE,2,pos + 1);
	new := CHR_TO_STRING(DWORD_TO_BYTE(HEX_TO_DWORD(seq)));
	URL_DECODE := REPLACE(URL_DECODE, new, 3, pos);
	pos := FIND(URL_DECODE,'%');
END_WHILE;


(* revision history
hm	27. apr. 2008	rev 1.0
	original version

hm	17. dec. 2008	rev 1.1
	changes name of function chr to chr_to_string

ks	10. mai. 2008	rev 1.2
	stringlength 250
*)

END_FUNCTION

// oscat_network/POUs/CO_NVERT/URL_ENCODE_1
FUNCTION URL_ENCODE_1 : STRING(STRING_LENGTH)
VAR_INPUT
	IN : STRING(STRING_LENGTH);
END_VAR
VAR
	pt_in : POINTER TO ARRAY[1..255] OF BYTE;
	pt_out : POINTER TO ARRAY[1..256] OF BYTE;
	pos_in : INT;
	pos_out : INT;
	stop : INT;
	tb : BYTE;
END_VAR


(*
version 1.1		10. may. 2010
programmer 	hugo
tested by		hugo

URL_ENCODE checks a string if it contains only non reserved characters for an url.
the non reserved characters are : [A..Z], [a..z], [0..9], -_.~
if reserved characters are found then these characters are converted to %HH while HH is the Hexadezimal representation of the character in Alphabetic Letters.
for example the reserved character # will be converted to '%23'.

*)

pt_in  := ADR(in);
pt_out := ADR(URL_ENCODE);

(* scan the input string and convert unallowed characters *)
pos_in := 1;
stop := LEN(in);
FOR pos_out := 1 TO 250 DO
	IF pos_in > stop THEN
		EXIT;
	ELSIF IS_URLCHR(pt_in^[pos_in]) THEN
		pt_out^[pos_out] := pt_in^[pos_in];
		(* increment in by 1 *)
		pos_in := pos_in + 1;
	ELSE
		(* cannot fit 3 digits, exit *)
		IF pos_out > 248 THEN EXIT; END_IF;
		(* invalid character that needs to be converted *)
		pt_out^[pos_out] := 37;    (* start with % sign *)
		pos_out := pos_out + 1;
		(* need to add the two hex digits *)
		tb := SHR(pt_in^[pos_in],4);
		IF tb > 9 THEN
			pt_out^[pos_out] := tb + 55;
		ELSE
			pt_out^[pos_out] := tb + 48;
		END_IF;
		pos_out := pos_out + 1;
		tb := pt_in^[pos_in] AND 16#0F;
		IF tb > 9 THEN
			pt_out^[pos_out] := tb + 55;
		ELSE
			pt_out^[pos_out] := tb + 48;
		END_IF;
		(* increment in and out because out has to move 3 digits *)
		pos_in := pos_in + 1;
	END_IF;
END_FOR;

(* terminate the output string *)
pt_out^[pos_out] := 0;

(* revision history
hm	27. apr. 2008	rev 1.0
	original version

ks	10. mai. 2008	rev 1.1
	stringlength 250

*)

END_FUNCTION

// oscat_network/POUs/CO_NVERT/URL_TO_STRING_1
FUNCTION URL_TO_STRING_1 : STRING(STRING_LENGTH)
VAR_INPUT
	IN : URL;
END_VAR


(*
version 1.1		10. may. 2010
programmer 	hugo
tested by		oscat

URL_TO_STRING generates a string from URL information suppied in IN..

*)

(*

http://hans:geheim@www.example.org:80/demo/example.cgi?land=de&stadt=aa#abschnitt1
|         |         |                  |                                |   |                                    |                                    |
|         |         |                 Host                         |   Pfad                            Query                           Anker
|         |         Passwort                                  Port
|        Benutzer
Protokoll

*)

(* attach protocol *)
IF IN.PROTOCOL <> '' THEN URL_TO_STRING := CONCAT(IN.PROTOCOL,'://'); END_IF;

(* attach user and password *)
IF IN.USER <> '' THEN
	URL_TO_STRING := CONCAT(URL_TO_STRING, IN.USER);
	IF IN.PASSWORD <> '' THEN
		URL_TO_STRING := CONCAT(URL_TO_STRING, ':');
		URL_TO_STRING := CONCAT(URL_TO_STRING, IN.PASSWORD);
	END_IF;
	URL_TO_STRING := CONCAT(URL_TO_STRING, '@');
END_IF;

(* attach domain *)
URL_TO_STRING := CONCAT(URL_TO_STRING, IN.DOMAIN);

(* attach Port *)
IF IN.PORT > 0 THEN
	URL_TO_STRING := CONCAT(URL_TO_STRING, ':');
	URL_TO_STRING := CONCAT(URL_TO_STRING, WORD_TO_STRING(IN.PORT));
END_IF;

(* attach path *)
URL_TO_STRING := CONCAT(URL_TO_STRING, IN.PATH);

(* attach query *)
IF IN.QUERY <> '' THEN
	URL_TO_STRING := CONCAT(URL_TO_STRING, '?');
	URL_TO_STRING := CONCAT(URL_TO_STRING, IN.QUERY);
END_IF;

(* attach anchor *)
IF IN.ANCHOR <> '' THEN
	URL_TO_STRING := CONCAT(URL_TO_STRING, '#');
	URL_TO_STRING := CONCAT(URL_TO_STRING, IN.ANCHOR);
END_IF;

(* revision history
hm	18. apr 2008	rev 1.0
	original version

ks	10. mai. 2008	rev 1.1
	stringlength 250
*)

END_FUNCTION

// oscat_network/POUs/DATA_LOG/DLOG_BOOL_1
FUNCTION_BLOCK DLOG_BOOL_1
VAR_IN_OUT
	X : DLOG_DATA;
END_VAR
VAR_INPUT
	STATE : BOOL;
	OFF : STRING;
	ON : STRING;
	COLUMN : STRING(40);
	DELTA : BOOL;
END_VAR
VAR_OUTPUT
END_VAR
VAR
	UCB : UNI_CIRCULAR_BUFFER;
	init : BOOL;
	id : WORD;
	last_delta : BOOL;
	state_last: BOOL;
END_VAR

(*
version 1.1		25. july. 2011
programmer		ks
tested by			ks

DLOG_BOOL legt den ON/OFF Text im FIFO-RING-Buffer ab um diesen mit den Baustein DLOG_STORE_*  aufzuzeichnen
*)

IF NOT init THEN
	init := TRUE;
	X.ID_MAX := X.ID_MAX + 1;
	id := WORD#16#0601; (* Quelltype BOOL , Zieltype STRING *)
END_IF;

IF X.ADD_HEADER THEN
	X.UCB.D_STRING := COLUMN;
	X.UCB.D_HEAD := id;
	X.UCB.D_MODE := 1;
	UCB(DATA:=X.UCB); (* Daten eintragen *)
ELSIF X.ADD_DATA THEN
	X.UCB.D_STRING := SEL(state_last,OFF,ON);
	X.UCB.D_HEAD := id;
	X.UCB.D_MODE := 1;
	UCB(DATA:=X.UCB); (* Daten eintragen *)
	last_delta := STATE;
ELSIF DELTA AND (STATE XOR last_delta) THEN
	X.ADD_DATA_REQ := TRUE;
	last_delta := STATE;
END_IF;
state_last := STATE;

(* revision history
ks	17. may. 2011	rev 1.0
	original version

ks	25. july.   2011	rev 1.1
	neue head information
*)

END_FUNCTION_BLOCK

// oscat_network/POUs/DATA_LOG/DLOG_DINT_1
FUNCTION_BLOCK DLOG_DINT_1
VAR_IN_OUT
	X : DLOG_DATA;
END_VAR
VAR_INPUT
	VALUE : DINT;
	COLUMN : STRING(40);
	DELTA : DINT;
END_VAR
VAR
	UCB : UNI_CIRCULAR_BUFFER;
	init : BOOL;
	id : WORD;
	delta_last : DINT;
	value_last : DINT;
END_VAR

(*
version 1.2		25. july. 2011
programmer		ks
tested by			ks

DLOG_DINT legt den DINT-Wert als STRING im FIFO-RING-Buffer ab um diesen mit den Baustein DLOG_STORE_* aufzuzeichnen
*)

IF NOT init THEN
	init := TRUE;
	X.ID_MAX := X.ID_MAX + 1;
	id := WORD#16#0801; (* Quelltype DINT , Zieltype STRING *)
END_IF;

IF X.ADD_HEADER THEN
	X.UCB.D_STRING := COLUMN;
	X.UCB.D_HEAD := id;
	X.UCB.D_MODE := 1;
	UCB(DATA:=X.UCB); (* Daten eintragen *)
ELSIF X.ADD_DATA THEN
	X.UCB.D_STRING := DINT_TO_STRING(value_last);
	X.UCB.D_HEAD := id;
	X.UCB.D_MODE := 1;
	UCB(DATA:=X.UCB); (* Daten eintragen *)
	delta_last := value_last;
ELSIF DELTA <> 0 THEN
	IF VALUE <= (delta_last - DELTA) OR VALUE >= (delta_last + DELTA) THEN
		X.ADD_DATA_REQ := TRUE;
		delta_last := VALUE;
	END_IF;
END_IF;
value_last := VALUE;

(* revision history
ks	01. jan. 2011	rev 1.0
	original version

ks	17. may. 2011	rev 1.1
	DELTA Funktion integriert

ks	25. july.   2011	rev 1.2
	neue head information
*)

END_FUNCTION_BLOCK

// oscat_network/POUs/DATA_LOG/DLOG_DT_1
FUNCTION_BLOCK DLOG_DT_1
VAR_IN_OUT
	X : DLOG_DATA;
END_VAR
VAR_INPUT
	FMT : STRING := '#A-#D-#H #N:#R:#T';
	COLUMN : STRING(40);
	DELTA : UDINT;
END_VAR

VAR_OUTPUT
END_VAR
VAR
	UCB : UNI_CIRCULAR_BUFFER;
	init : BOOL;
	id : WORD;
	delta_last : DT;
END_VAR

(*
version 1.2		25. july. 2011
programmer		ks
tested by			ks

DLOG_DT legt den formatierten DT String im FIFO-RING-Buffer ab um diesen mit den Baustein DLOG_STORE_*  aufzuzeichnen
*)

IF NOT init THEN
	init := TRUE;
	X.ID_MAX := X.ID_MAX + 1;
	id := WORD#16#0D01; (* Quelltype DT , Zieltype STRING *)
END_IF;

IF X.ADD_HEADER THEN
	X.UCB.D_STRING := COLUMN;
	X.UCB.D_HEAD := id;
	X.UCB.D_MODE := 1;
	UCB(DATA:=X.UCB); (* Daten eintragen *)
ELSIF X.ADD_DATA THEN
	X.UCB.D_STRING := DT_TO_STRF(DTI:=X.DTI,MS:=0,FMT:=FMT,LANG:=0);
	X.UCB.D_HEAD := id;
	X.UCB.D_MODE := 1;
	UCB(DATA:=X.UCB); (* Daten eintragen *)
	delta_last := X.DTI;
ELSIF DELTA <> 0 THEN
	IF DT_TO_UDINT(X.DTI) >= (DT_TO_UDINT(delta_last) + DELTA) THEN
		X.ADD_DATA_REQ := TRUE;
		delta_last := X.DTI;
	END_IF;
END_IF;

(* revision history
ks	01. jan. 2011	rev 1.0
	original version

ks	17. may. 2011	rev 1.1
	COLUMN STRING(40), delta

ks	25. july.   2011	rev 1.2
	neue head information
*)

END_FUNCTION_BLOCK

// oscat_network/POUs/DATA_LOG/DLOG_FILE_TO_FTP_1
FUNCTION_BLOCK DLOG_FILE_TO_FTP_1
VAR_IN_OUT
	X : DLOG_DATA;
END_VAR
VAR_INPUT
	FTP_URL : STRING(STRING_LENGTH);
	FTP_ACTIV : BOOL;
	FILE_DELETE : BOOL;
	TIMEOUT : TIME := T#30s;
	RETRY : INT;
	RETRY_TIME : TIME := T#30s;
	DNS_IP4 : DWORD;
	PLC_IP4 : DWORD;
END_VAR
VAR_OUTPUT
	DONE : BOOL;
	BUSY : BOOL;
	ERROR_C : DWORD;
	ERROR_T : BYTE;
END_VAR
VAR
	UCBD : UNI_CIRCULAR_BUFFER_DATA;
	UCB : UNI_CIRCULAR_BUFFER;
	FTP_CLIENT : FTP_CLIENT;
	WT_1 : TON;
	ftrig_old : BOOL;
	filename : STRING;
	step : INT;
	ftp_busy : BOOL;
	ftp_done : BOOL;
	cnt : INT;

	(*LOG_MSG : LOG_MSG;
	_debug_enable : BOOL := TRUE;*)
END_VAR

(*
version 1.1		26. july. 2011
programmer		ks
tested by			ks

DLOG_FILE_TO_FTP der Baustein kopiert bzw verschiebt die vom DLOG_STORE_FILE_CSV erzeugten Dateien auf einem FTP-Server
*)

(* neue Filenamen speichern *)
IF X.NEW_FILE_RTRIG AND ftrig_old = FALSE THEN
	UCBD.D_HEAD := 1;
	UCBD.D_MODE := 1;
	UCBD.D_STRING := X.NEW_FILE;
	UCB(DATA:=UCBD); (* Daten eintragen *)
END_IF;
ftrig_old := X.NEW_FILE_RTRIG;

CASE step OF

00:	IF UCBD.BUF_COUNT > 0 AND ftp_busy = FALSE THEN
		UCBD.D_MODE := 12; (* Daten lesen und löschen *)
		UCB(DATA:=UCBD);
		filename := UCBD.D_STRING;
		cnt := 0;
		step := 10;
	END_IF;

10:	IF ftp_busy = FALSE THEN
		IF ftp_done THEN
			(*####################  DEBUG-MESSAGE  ###################################*)
			(*IF _debug_enable THEN
				LOG_CL.NEW_MSG := 'F_T_FTP: /FILE OK >~1<';
				LOG_CL.PRINTF[1] := filename;
				LOG_MSG();
			END_IF;*)
			(*########################################################################*)
			step := 0;
		ELSE
			step := 20; (* pause nach error *)
		END_IF;
	END_IF;

20:	IF WT_1.Q THEN (* Wartezeit *)
		cnt := cnt - 1;
		IF RETRY = 0 THEN (* FTP Transfer unbegrenzt wiederholen *)
			(*####################  DEBUG-MESSAGE  ###################################*)
			(*IF _debug_enable THEN
				LOG_CL.NEW_MSG := 'F_T_FTP: Auftrag unbegrenzt wiederholen /file: ~2';
				LOG_CL.PRINTF[2] := filename;
				LOG_MSG();
			END_IF;*)
			(*########################################################################*)
			step := 10; (* FTP Transfer wiederholen *)
		ELSIF cnt >= 0 THEN
			(*####################  DEBUG-MESSAGE  ###################################*)
			(*IF _debug_enable THEN
				LOG_CL.NEW_MSG := 'F_T_FTP: Auftrag wiederholen /cnt: ~1 /file: ~2';
				LOG_CL.PRINTF[1] := INT_TO_STRING(cnt);
				LOG_CL.PRINTF[2] := filename;
				LOG_MSG();
			END_IF;*)
			(*########################################################################*)
			step := 10; (* FTP Transfer wiederholen *)
		ELSE
			(*####################  DEBUG-MESSAGE  ###################################*)
			(*IF _debug_enable THEN
				LOG_CL.NEW_MSG := 'F_T_FTP: Auftrag verworfen /file: ~2';
				LOG_CL.PRINTF[2] := filename;
				LOG_MSG();
			END_IF;*)
			(*########################################################################*)
			step := 0; (* FTP Auftrag verwerfen *)
		END_IF;
	END_IF;

END_CASE;

BUSY := step = 10;
DONE := step = 0;
WT_1(IN:= step = 20, PT:= RETRY_TIME);

FTP_CLIENT(
	ACTIVATE:= BUSY,
	FILENAME:= filename,
	FTP_URL:= FTP_URL,
	FTP_DOWNLOAD:= FALSE,
	FTP_ACTIV:= FTP_ACTIV,
	FILE_DELETE:= FILE_DELETE,
	TIMEOUT:= TIMEOUT,
	DNS_IP4:= DNS_IP4,
	PLC_IP4:= PLC_IP4,
	DONE=> ftp_done,
	BUSY=> ftp_busy,
	ERROR_C=> ERROR_C,
	ERROR_T=> ERROR_T
	);

(* revision history
ks	01. jan. 2011	rev 1.0
	original version

ks	26. july. 2011	rev 1.1
	codeoptimierung D_MODE 12
*)

END_FUNCTION_BLOCK

// oscat_network/POUs/NETWORK/LOG_MSG
FUNCTION_BLOCK LOG_MSG
(* VAR_EXTERNAL
	LOG_CL :	LOG_CONTROL;
END_VAR *)
VAR
	FB_PRINT_SF :PRINT_SF;
	idX : INT;
END_VAR

(*
version 1.0		01 mai 2010
programmer		ks
tested by		ks

LOG_MSG trägt Meldungen in den Loggingbuffer ein
*)

IF DWORD_TO_BYTE(SHL(LOG_CL.NEW_MSG_OPTION,16)) > LOG_CL.LEVEL THEN RETURN; END_IF; (* Logging freigegeben ?*)

FB_PRINT_SF(PRINTF_DATA := LOG_CL.PRINTF,STR := LOG_CL.NEW_MSG);

IF LOG_CL.RESET THEN (* Logeinträge löschen *)
	LOG_CL.RESET := FALSE;
	LOG_CL.RING_MODE := FALSE;
	LOG_CL.IDX := 0;
	LOG_CL.UPDATE_COUNT := LOG_CL.UPDATE_COUNT + UINT#1; (* UpdateCount erhöhen *)
END_IF;

IF LOG_CL.SIZE > 0 THEN (* size wert ist eingetragen *)
	IF LEN(LOG_CL.NEW_MSG) > 0 THEN (* Meldung in Puffer eintragen *)
		IF (LOG_CL.IDX >= LOG_CL.SIZE) THEN
			LOG_CL.RING_MODE := TRUE; (* bei Überlauf = Ringbuffermodus *)
			LOG_CL.IDX := 0; (* wieder auf arrayanfang positionieren *)
		END_IF;

		LOG_CL.UPDATE_COUNT := LOG_CL.UPDATE_COUNT + UINT#1; (* UpdateCount erhöhen *)
		LOG_CL.IDX := LOG_CL.IDX + INT#1; (* nächste freie Position *)
		idx := LOG_CL.IDX; (* lade aktuelle Log-Puffer Positition *)
		LOG_CL.MSG[idx] := LOG_CL.NEW_MSG; (* neuen Log-String in puffer ablegen  *)
		LOG_CL.MSG_OPTION[idx] := LOG_CL.NEW_MSG_OPTION; (* neue Log-String Option in puffer ablegen  *)
		LOG_CL.NEW_MSG := ''; (* letzten Log-String löschen *)
	END_IF;
END_IF;

END_FUNCTION_BLOCK

// oscat_network/POUs/NETWORK/PRINT_SF
FUNCTION_BLOCK PRINT_SF
VAR_IN_OUT
	PRINTF_DATA : PRINTF_DATA;
	STR : STRING(LOG_SIZE);
END_VAR
VAR
	pos : INT;
	c : INT;
	src : STRING(1) := '~';
	run : BOOL;
END_VAR

(*

version 1.0 		14. aug. 2009
programmer 	ks
tested by		ks

PRINTF erzeugt aus einem Parameterstring und den übergebenen Parameterdaten einen Text
*)

IF LEN(STR) > 0 THEN
	run := TRUE;

	WHILE (run) DO
		pos := FIND(STR,src);
		PRINTF_DATA[10] := '';

		IF pos = 0 THEN
			run:= FALSE;
		ELSE
			c := CODE(STR:=STR,POS:=pos + 1);
			IF ISC_NUM(INT_TO_BYTE(c)) THEN
				c := c - 48; (* notwendig weil innerhalb einer indexangabe nur eine var stehen darf *)
				PRINTF_DATA[10] := PRINTF_DATA[c]; (* Kommando 1-9 ergibt Parameterindex 1-9 *)
				(* Parameter gegen Text tauschen *)
			END_IF;
			IF LEN(PRINTF_DATA[10]) + LEN(STR) > LOG_SIZE THEN
				PRINTF_DATA[10] := '..';
			END_IF;
			(* pcworx: aus und eingangsstring muss verschieden sein *)
			PRINTF_DATA[11] := STR;
			STR := REPLACE(PRINTF_DATA[11],PRINTF_DATA[10],2,pos);
		END_IF;
	END_WHILE;
END_IF;

(* revision history

ks	14. aug. 2009	rev 1.0
	original version

*)

END_FUNCTION_BLOCK

// oscat_network/POUs/NETWORK/FTP_CLIENT
FUNCTION_BLOCK FTP_CLIENT
VAR_INPUT
	ACTIVATE : BOOL;
	FILENAME : STRING;
	FTP_URL : STRING(STRING_LENGTH);
	FTP_DOWNLOAD : BOOL;
	FTP_ACTIV : BOOL;
	FILE_DELETE : BOOL;
	TIMEOUT : TIME;
	DNS_IP4 : DWORD;
	PLC_IP4 : DWORD;
END_VAR
VAR_OUTPUT
	DONE : BOOL;
	BUSY : BOOL;
	ERROR_C : DWORD;
	ERROR_T : BYTE;
END_VAR
VAR
	IP_C1 : IP_C; (* IP_Control Verwaltungsstruktur *)
	IP_C2 : IP_C; (* IP_Control Verwaltungsstruktur *)
	S_BUF1 : NETWORK_BUFFER;
	S_BUF2 : NETWORK_BUFFER;
	R_BUF1 : NETWORK_BUFFER;
	R_BUF2 : NETWORK_BUFFER;
	URL_DATA : url;
	DNS_CLIENT : DNS_CLIENT;
	IPC1 : IP_CONTROL;
	IPC2 : IP_CONTROL;
	FS : FILE_SERVER;
	FSD : FILE_SERVER_DATA;

	activate_last : BOOL;
	step : INT;
	snd_step : INT;
	snd_text :	STRING(STRING_LENGTH);
	rcv_text :	STRING(STRING_LENGTH);
	rcv_state : INT;
	TON_WAIT : TON;
	last_step : INT;
	next_step : INT;
	idx1 : INT;
	idx2 : INT;
	str1 : STRING(STRING_LENGTH);
	str2 : STRING(STRING_LENGTH);
	ftp_path : STRING;
	byar : ARRAY [0..5] OF BYTE;
	dw_tmp : DWORD;
	w_tmp : WORD;
	fpd : FILE_PATH_DATA;
	timeout2 : TIME;
	timeout3 : TIME;
	ftp_file_size : UDINT;
	ip_c1_red_disable : BOOL; (* IP_CONTROL 1 - Remote Disconnect Error unterdrücken *)
	ip_c2_red_disable : BOOL; (* IP_CONTROL 1 - Remote Disconnect Error unterdrücken *)

	(*LOG_MSG : LOG_MSG;
	_debug_enable : BOOL := FALSE;*)

END_VAR
(*
version 1.2		11.may 2011
programmer		ks
tested by			ks

FTP_CLIENT dient zum senden und empfangen von dateien von einem FTP-Server.



110 Restart marker reply 										Markierung für Wiederaufnahme der Übertragung 
120 Service ready in x minutes 									Dienst steht in x Minuten zu Verfügung 
125 Data connection already open; 								transfer starting Datenverbindung besteht bereits; beginne mit der Übertragung 
150 File status okay; about to open data connection 					Dateistatus OK; Datenverbindung wird aufgebaut 
200 Command okay 											Befehl OK 
202 Command not implemented 									Befehl nicht implementiert 
211   														Antwort für Systemstatus oder Hilfefunktion des Systems 
212   														Verzeichnisstatus 
213   														Dateistatus 
214   														Meldung der Hilfefunktion 
215 NAME system type 										Angabe des Systemtyps 
220 Service ready for new user 									Dienst bereit für neuen Benutzer 
221 Service closing control connection 							Steuerverbindung des Dienstes wird getrennt; Benutzer wird abgemeldet 
225 Data connection open; no transfer in progress 					Datenverbindung hergestellt; derzeit keine Übertragung 
226 Closing data connection. Requested file action successful 		Datenverbindung wird getrennt 
227 Entering Passive Mode 										Passiver Modus aktiviert 
230 User logged in, proceed 									Benutzer angemeldet, bitte fortfahren 
250 Requested file action okay, completed 						Angeforderter Vorgang OK, beendet 
257 "PATH" created 											"PFAD" wurde erstellt 
331 User name okay, need password 							Benutzername OK, Kennwort erforderlich 
332 Need account for login 										Benutzerkonto zur Anmeldung erforderlich 
350 Requested file action pending further information 				Mehr Informationen für Dateivorgang erforderlich 
421 Service not available, closing control connection 				Dienst nicht verfügbar, Steuerverbindung wird getrennt 
425 Can't open data connection 									Datenverbindung kann nicht hergestellt werden 
426 Connection closed; transfer aborted Verbindung getrennt; 		Übertragung abgebrochen 
450 Requested file action not taken; File unavailable 				Angeforderter Dateivorgang wurde nicht ausgeführt; Datei nicht verfügbar 
451 Requested action aborted: local error in processing 				Angeforderter Vorgang abgebrochen: Lokaler Fehler bei der Bearbeitung 
452 Requested action not taken; Insufficient storage space in system 	Angeforderter Vorgang nicht ausgeführt; Nicht genügend Speicherplatz auf System 
500 Syntax error 												Befehl nicht erkannt 
501 Syntax error in parameters or arguments 						Syntaxfehler bei den Parametern 
502 Command not implemented 									Befehl nicht implementiert 
503 Bad sequence of commands 								Ungültige Befehlsabfolge 
504 Command not implemented for that parameter 					Befehl für diesen Parameter nicht implementiert 
530 Not logged in 												Nicht angemeldet 
532 Need account for storing files 								Zum Speichern von Dateien Anmeldung erforderlich 
550 Requested file action not taken; File unavailable Angeforderter 	Dateivorgang wurde nicht ausgeführt; Datei nicht verfügbar 
551 Requested action aborted: page type unknown 					Angeforderter Vorgang abgebrochen: Unbekannter Seitentyp 
552 Requested file action aborted: Exceeded storage allocation 		Angeforderter Dateivorgang abgebrochen: Nicht genügend Platz in aktuellem Verzeichnis oder Datensatz 
553 Requested action not taken: File name not allowed 				Angeforderter Vorgang nicht ausgeführt: Unzulässiger Dateiname 

#########################
ERROR_T

1 = DNS_CLIENT
2 = FTP Steuerkanal
3 = FTP Datenkanal
4 = FILE_SERVER
5 = Ablaufstörung
#########################

*)

CASE step OF

00:	IF ACTIVATE AND NOT activate_last THEN
		ftp_file_size := UDINT#0;
		TIMEOUT := MAX(T#10s,TIMEOUT);
		timeout2 := TIMEOUT + T#1s;
		timeout3 := TIMEOUT / 2;
		DONE := FALSE;
		ip_c1_red_disable := FALSE;
		ip_c2_red_disable := FALSE;
		ERROR_C := DWORD#0;
		ERROR_T := BYTE#0;
		FSD.ERROR := BYTE#0;
		URL_DATA := STRING_TO_URL(STR:=FTP_URL,DEFAULT_PROTOCOL:='',DEFAULT_PATH:='/');
		IF LEN(URL_DATA.USER) = 0 THEN
			URL_DATA.USER := 'Anonymous';
			URL_DATA.PASSWORD := 'User@';
		END_IF;

		FILE_PATH_SPLIT(FILENAME:=FILENAME,X:=fpd); (* Datei-Path zerlegen *)
		str1 := fpd.FILENAME; (* zwischenspeichern *)
		FILE_PATH_SPLIT(FILENAME:=URL_DATA.PATH,X:=fpd); (* FTP-Path zerlegen *)
		IF LEN(fpd.FILENAME) = 0 THEN (* wenn FTP-Path keinen Dateinamen enthält , dann den Namen der lokalen Datei benutzen *)
			ftp_path := CONCAT(URL_DATA.PATH,str1);
		ELSE
			ftp_path := URL_DATA.PATH;
		END_IF;
		step := 10;
	END_IF;

10:	IF DNS_CLIENT.DONE THEN
		step := 20;
	ELSIF DNS_CLIENT.ERROR <> DWORD#0 THEN
		ERROR_C := DNS_CLIENT.ERROR;
		ERROR_T := BYTE#1;
		step := 980;
	END_IF;

20:	(* FTP Steuerkanal einrichten *)
	IP_C1.C_PORT := WORD#21; (* Portnummer eintragen *)
  	IP_C1.C_IP := DNS_CLIENT.IP4; (* IP eintragen *)
  	IP_C1.C_MODE := BYTE#0; (* Mode: TCP+ACTIV+PORT *)
  	IP_C1.TIME_RESET := TRUE; (* Zeitueberwachung rücksetzen *)
  	IP_C1.C_ENABLE := TRUE; (* Verbindungsaufbau freigeben *)
  	IP_C1.R_OBSERVE := TRUE; (* Empfangsueberwachung *)
	R_BUF1.SIZE := UINT#0;

  	IP_C2.C_ENABLE   := FALSE; (* Verbindungsaufbau sperren *)
	step := 30;

30:	IF rcv_state = 220 THEN (* 220 = Service ready for new user *)
		snd_text := CONCAT('USER ',URL_DATA.USER);
		next_step := 40;
	END_IF;

40:	IF rcv_state = 331 THEN (* 331 = User name okay, need password *)
		snd_text := CONCAT('PASS ',URL_DATA.PASSWORD);
		next_step := 50;
	ELSIF rcv_state = 230 THEN (* 230 = User logged in, proceed *)
		next_step := 50;
	ELSIF rcv_state = 220 THEN (* 220 = Service ready for new user *)
		next_step := 20; (* WORK verbindung sollte ab/aufgebaut werden *)
	END_IF;

50:	IF rcv_state = 230 THEN (* 230 = User logged in, proceed *)
		snd_text := 'TYPE I';  (* binären Modus aktivieren *)
		next_step := 54;
	END_IF;

54:	IF rcv_state = 200 THEN (* 200 = Command okay *)
		IF FTP_DOWNLOAD THEN (* Datei von FTP Empfangen *)
			snd_text := CONCAT('SIZE ', ftp_path); (* SIZE /PFAD/FILENAME *)
			next_step := 56;
		ELSE
			step := 60;
		END_IF;
	END_IF;

56:	IF rcv_state = 213 THEN (* 213 Filesize *)
		str1 := ELEMENT_GET(SEP:=BYTE#32,POS:=1,ELEMENT:=rcv_text);
		ftp_file_size := STRING_TO_UDINT(str1); (* Dateigroesse in bytes gestimmen *)
		step := 60;
	END_IF;

60:	IF FTP_ACTIV THEN (* FTP Server aktiv *)
		IF URL_DATA.PORT = WORD#0 THEN
			URL_DATA.PORT := WORD#20; (* Standard Datenkanal *)
		END_IF;
		str2 := '';
		dw_tmp := PLC_IP4;
		FOR idx1 := 0 TO 5 DO
			IF idx1 = 4 THEN
				dw_tmp := ROR(WORD_TO_DWORD(URL_DATA.PORT),8);
			ELSE
				dw_tmp := ROL(dw_tmp,8);
			END_IF;
			str2 := CONCAT(str2,BYTE_TO_STRING(DWORD_TO_BYTE(dw_tmp)));
			IF idx1 < 5 THEN
				str2 := CONCAT(str2,',');
			END_IF;
		END_FOR;
		dw_tmp := DNS_CLIENT.IP4; (* IP eintragen *)
		w_tmp := URL_DATA.PORT; (* Port Nummer des Datenkanals *)
		snd_text := CONCAT('PORT ',str2); (* FTP Server in den aktiv-mode schalten *)
		next_step := 80;
	ELSE
		snd_text := 'PASV';  (* FTP Server in den passiv-mode schalten *)
		next_step := 70;
	END_IF;
	step := 999; (* Warten auf next_step *)

70:	IF rcv_state = 227 THEN (* 227 = Entered Passive Mode (213,202,225,43,212,186) *)
		idx1 := FIND(rcv_text , '(' );
		idx2 := FIND(rcv_text , ')' );
		IF idx1 > 0 AND idx2 > idx1+1 THEN
			str1 := MID(rcv_text, idx2 - idx1 - 1, idx1+1);
			FOR idx1 := 0 TO 5 DO
				str2 := ELEMENT_GET(SEP:=BYTE#44,POS:=idx1,ELEMENT:=str1);
				byar[idx1] := STRING_TO_BYTE(str2);
			END_FOR;
			dw_tmp := DWORD_OF_BYTE(byar[0],byar[1],byar[2],byar[3]); (* IP Adresse des Datenkanals *)
			w_tmp := WORD_OF_BYTE(byar[4],byar[5]); (* Port Nummer des Datenkanals *)
		END_IF;
		step := 100;
	END_IF;

80:	IF rcv_state = 200 THEN (* 200 = PORT command successful *)
		step := 100;
	END_IF;

100:IP_C2.C_MODE := SEL(FTP_ACTIV,BYTE#0,BYTE#2); (* Aktiv = Mode 2: TCP+PASSIV+PORT / passiv = Mode 0: TCP+ACTIV+PORT *)
	IP_C2.C_IP := dw_tmp; (* IP Adresse des Datenkanals *)
	IP_C2.C_PORT := w_tmp; (* Port Nummer des Datenkanals *)
  	IP_C2.TIME_RESET := TRUE; (* Zeitueberwachung rücksetzen *)
  	IP_C2.C_ENABLE := TRUE; (* Verbindungsaufbau freigeben *)
	IP_C2.R_OBSERVE := FALSE; (* Empfangsueberwachung *)
	R_BUF2.SIZE := UINT#0;
	step := 120;

120:IF IP_C2.C_STATE > BYTE#127 THEN (* FTP Datenkanal aufgebaut *)
		IF FTP_DOWNLOAD THEN (* File von FTP empfangen *)
			IP_C2.MAILBOX[3] := BYTE#1; (* IP Empfang sperren *)
			step := 400;
		ELSE
			snd_text := 'STOR ';
			next_step := 140;
			snd_text := CONCAT(snd_text, ftp_path); (* STORE /PFAD/FILENAME *)
			step := 999; (* Warten auf next_step *)
		END_IF;
	END_IF;

(* ============== File an FTP senden ================ *)

140:IF rcv_state = 125 OR rcv_state = 150 THEN (* 125 = Data connection already open / 150 = File status okay; about to open data connection *)
		step := 160;
	END_IF;

160:FSD.FILENAME := FILENAME; (* Dateiname *)
	FSD.MODE := BYTE#1; (* vorhandene Datei zum lesen öffnen *)
	FSD.OFFSET := UDINT#0; (* Start bei Dateianfang *)
	FSD.AUTO_CLOSE := T#0s; (* kein Auto-Close verwenden *)
	S_BUF2.SIZE := UINT#65535; (* maximale länge einlesen *)
	IP_C2.MAILBOX[2] := BYTE#1; (* IP Senden blockieren *)
	step := 200;

200:IF FSD.MODE = BYTE#0 AND FSD.ERROR = BYTE#0 THEN
		IP_C2.MAILBOX[2] := BYTE#0; (* IP Senden erlauben *)
		step := 210;
	END_IF;

210:IF S_BUF2.SIZE = UINT#0 THEN (* warten bis alle daten gesendet sind *)
		IF FSD.FILE_SIZE - FSD.OFFSET > UDINT#0 THEN
			FSD.MODE := BYTE#1; (* vorhandene Datei zum lesen öffnen *)
			S_BUF2.SIZE := UINT#65535; (* maximale länge einlesen *)
			IP_C2.MAILBOX[2] := BYTE#1; (* IP Senden blockieren *)
			step := 200;
		ELSE
			IP_C2.C_ENABLE := FALSE; (* FTP Datenkanal schliessen *)
			step := 300;
		END_IF;
	END_IF;

300:IF rcv_state = 226 THEN (* 226 Closing data connection. Requested file action successful  *)
		snd_text := 'QUIT';
		ip_c1_red_disable := TRUE;
		next_step := 320;
	END_IF;

320:IF rcv_state = 221 OR TON_WAIT.ET > timeout3  THEN (* 221 Service closing control connection *)
		IP_C1.C_ENABLE := FALSE; (* FTP Steuerkanal schliessen *)
		IF FILE_DELETE THEN (* Datei nach transfer löschen *)
			FSD.MODE := BYTE#4; (* File Remove *)
			step := 340;
		ELSE
			step := 900;
		END_IF;
	END_IF;

340:IF FSD.MODE = BYTE#0 AND FSD.ERROR = BYTE#0 THEN
		step := 900;
	END_IF;

(*  ============== File vom FTP Empfangen  ============== *)

400:snd_text := 'RETR ';
	next_step := 410;
	snd_text := CONCAT(snd_text, ftp_path); (* RETR /PFAD/FILENAME *)
	step := 999; (* Warten auf next_step *)

410:IF rcv_state = 125 OR rcv_state = 150 THEN (* 125 = Data connection already open / 150 = File status okay; about to open data connection *)
		IP_C2.R_OBSERVE := TRUE; (* Empfangsueberwachung *)
		step := 420;
	END_IF;

420:FSD.FILENAME := FILENAME; (* Dateiname *)
	FSD.MODE := BYTE#3; (* Datei neu anlegen *)
	FSD.OFFSET := UDINT#0; (* Start bei Dateianfang *)
	FSD.AUTO_CLOSE := T#0s; (* kein Auto-Close verwenden *)
	step := 460;

440:IF R_BUF2.SIZE > UINT#0 THEN (* warten bis daten empfangen wurden *)
		IP_C2.MAILBOX[3] := BYTE#1; (* IP Empfang blockieren bis Daten in Datei geschrieben wurden *)
		FSD.MODE := BYTE#3; (* Daten in Datei schreiben *)
		step := 460;
	ELSIF FSD.FILE_SIZE = ftp_file_size THEN (* Verbindung abgebaut ? , oder 226 = Closing data connection. Requested file action successful *)
		IP_C2.C_ENABLE := FALSE; (* FTP Datenkanal schliessen *)
		ip_c2_red_disable := TRUE;
		step := 700;
	END_IF;

460:IF FSD.MODE = BYTE#0 AND FSD.ERROR = BYTE#0 THEN (* warten bis Daten geschreiben wurden *)
		R_BUF2.SIZE := UINT#0; (* Daten löschen *)
		IP_C2.MAILBOX[3] := BYTE#0; (* IP Empfang wieder erlauben *)
		step := 440;
	END_IF;

(* ================================================== *)

700:IF rcv_state = 226 OR  TON_WAIT.ET > timeout3 THEN (* 226 Closing control connection. Requested file action successful  *)
		IF FTP_DOWNLOAD AND FILE_DELETE THEN (* FTP Download und File löschen ? *)
			snd_text := CONCAT('DELE ', ftp_path); (* DELE /PFAD/FILENAME *)
			next_step := 720;
		ELSE
			step := 740;
		END_IF;
	END_IF;

720:IF rcv_state = 250 THEN (* 250 Requested file action okay, completed *)
		step := 740;
	END_IF;

740:snd_text := 'QUIT';
	ip_c1_red_disable := TRUE;
	next_step := 760;
	step := 999; (* Warten auf next_step *)

760:IF rcv_state = 221 OR TON_WAIT.ET > timeout3 THEN (* 221 Service closing control connection  *)
		IP_C1.C_ENABLE := FALSE; (* FTP Steuerkanal schliessen *)
		IF NOT FTP_DOWNLOAD AND FILE_DELETE THEN (* FTP Upload und Datei nach transfer löschen *)
			FSD.MODE := BYTE#4; (* File Remove *)
			step := 780;
		ELSE
			step := 900;
		END_IF;
	END_IF;

780:IF FSD.MODE = BYTE#0 AND FSD.ERROR = BYTE#0 THEN
		step := 900;
	END_IF;

(* ================================================== *)

900:DONE := TRUE;
	step := 980;

980:IP_C1.C_ENABLE := FALSE; (* FTP Steuerkanal schliessen *)
	IP_C2.C_ENABLE := FALSE; (* FTP Datenkanal schliessen *)
	IP_C2.MAILBOX[2] := BYTE#0; (* IP Senden wieder erlauben *)
	IP_C2.MAILBOX[3] := BYTE#0; (* IP Empfang wieder erlauben *)
	S_BUF1.SIZE := UINT#0;
	S_BUF2.SIZE := UINT#0;
	R_BUF1.SIZE := UINT#0;
	R_BUF2.SIZE := UINT#0;
	ftp_file_size := UDINT#0;
	snd_step := 0;
	next_step := 0;
	FSD.MODE := BYTE#5; (* Datei schliessen *)
	step := 990;

990:IF IP_C1.C_STATE = BYTE#0 AND IP_C2.C_STATE = BYTE#0 AND FSD.FILE_OPEN = FALSE THEN
		step := 0;
	END_IF;

999: ; (* Dummy Schritt, warten bis neuer schritt durch "next_step" aktiv wird *)

END_CASE;

(* ++++++++++++++++++++++++++++++++++++++++++++++++++++++++++ *)

IF step >= 30 THEN
	IF R_BUF1.SIZE > UINT#0 THEN (* Daten wurden empfangen ? *)
		idx1 := UINT_TO_INT(R_BUF1.SIZE);
		REPEAT (* zeilenterminierung erkennen und echtes TEXT-Ende bestimmen *)
			idx1 := idx1 - 1;
		UNTIL idx1 = 0 OR R_BUF1.BUFFER[idx1] >= BYTE#32 (* TRUE = EXIT *)
		END_REPEAT;
		idx1 := idx1 + 1; (* index auf SIZE umrechnen *)
		rcv_text := BUFFER_TO_STRING(PT:=ADR(R_BUF1.BUFFER),SIZE:=idx1,START:=0,STOP:=STRING_LENGTH-1);
		IF LEN(rcv_text) >= 3 THEN (* Statuscode prüfen und auswerten *)
			str1 := LEFT(rcv_text,3);
			IF IS_NUM(STR:=str1) THEN (* enthält nur Zahlen ? *)
				rcv_state := STRING_TO_INT(str1);
			END_IF;
			IP_C1.R_OBSERVE := FALSE;
		END_IF;
		R_BUF1.SIZE := UINT#0; (* daten löschen *)

	        (*####################  DEBUG-MESSAGE  ###################################*)
	        (*IF _debug_enable THEN
	          LOG_CL.NEW_MSG := 'RCV: >~1<';
	          LOG_CL.PRINTF[1] := rcv_text;
	          LOG_MSG();
	        END_IF;*)
	        (*########################################################################*)

	END_IF;
END_IF;

(* automatisches Datensenden *)

CASE snd_step OF

00:	IF LEN(snd_text) > 0 THEN
	        (*####################  DEBUG-MESSAGE  ###################################*)
	        (*IF _debug_enable THEN
	          LOG_CL.NEW_MSG := 'SND: >~1<';
	          LOG_CL.PRINTF[1] := snd_text;
	          LOG_MSG();
	        END_IF;*)
	        (*########################################################################*)
		_STRING_TO_BUFFER(str:=snd_text,pos:=0,pt:=ADR(S_BUF1.BUFFER),size:=SIZEOF(S_BUF1.BUFFER)); (* String in puffer kopieren *)
		idx1 := LEN(snd_text);
		S_BUF1.BUFFER[idx1] := BYTE#16#0D;
		idx1 := idx1 + 1;
		S_BUF1.BUFFER[idx1] := BYTE#16#0A;
		idx1 := idx1 + 1;
		S_BUF1.SIZE := INT_TO_UINT(idx1); (* Sendelänge eintragen *)
		R_BUF1.SIZE := UINT#0; (* Empfangsbuffer rücksetzen *)
		IP_C1.R_OBSERVE := TRUE;
		rcv_state := 9999; (* letzen FTP Status löschen *)
		snd_text := '';
		snd_step := 10;
	END_IF;

10:	IF S_BUF1.SIZE = UINT#0 THEN (* warten bis alle daten gesendet sind *)
		step := next_step;
		snd_step := 0;
	END_IF;

END_CASE;

(* Globale Fehlerbehandlung für Haupt-Routine *)
IF ERROR_T = BYTE#0 AND step > 20 THEN (* noch kein Fehler gespeichert und Hauptroutine aktiv *)

	IF IP_C1.ERROR > DWORD#0 AND IP_C1.C_ENABLE AND NOT IP_C1.TIME_RESET THEN  (* IP Control 1 *)
		IF ip_c1_red_disable = FALSE OR IP_C1.ERROR <> DWORD#16#FD000000 THEN
			ERROR_C := IP_C1.ERROR;
			ERROR_T := BYTE#2;
			step := 980;
		END_IF;
	END_IF;

	IF IP_C2.ERROR > DWORD#0 AND IP_C2.C_ENABLE AND NOT IP_C2.TIME_RESET THEN  (* IP Control 2 *)
		IF ip_c2_red_disable = FALSE OR IP_C2.ERROR <> DWORD#16#FD000000 THEN
			ERROR_C := IP_C2.ERROR;
			ERROR_T := BYTE#3;
			step := 980;
		END_IF;
	END_IF;

	IF FSD.MODE = BYTE#0 THEN
		IF FSD.ERROR > BYTE#0 THEN
			ERROR_C := BYTE_TO_DWORD(FSD.ERROR);
			ERROR_T := BYTE#4; (* Dateizugriff *)
			step := 980;
		END_IF;
	END_IF;
END_IF;

IF TON_WAIT.Q THEN (* Ablaufstörung - Schrittkette *)
	ERROR_C := SHL(INT_TO_DWORD(step),16) OR INT_TO_DWORD(rcv_state); (* aktuellen Schritt und letzten FTP Status eintragen *)
	ERROR_T := BYTE#5;
	step := 980;
END_IF;

(* ######################################################## *)

DNS_CLIENT(IP_C:=IP_C1, S_BUF:=S_BUF1, R_BUF:=R_BUF1, DOMAIN:=URL_DATA.DOMAIN, IP4_DNS:= DNS_IP4, ACTIVATE:=step=10); (* DNS-Client *)
IPC1(IP:= DWORD#0, PORT:= WORD#0 , TIME_OUT:= TIMEOUT, IP_C:= IP_C1, S_BUF:= S_BUF1, R_BUF:= R_BUF1); (* FTP Steuerkanal *)
IPC2(IP:= DWORD#0, PORT:= WORD#0 , TIME_OUT:= TIMEOUT, IP_C:= IP_C2, S_BUF:= S_BUF2, R_BUF:= R_BUF2); (* FTP Datenkanal *)

TON_WAIT(IN:=step = last_step AND step > 0,PT:=timeout2);
last_step := step;
activate_last := ACTIVATE;
BUSY := step <> 0;

IF FTP_DOWNLOAD THEN (* FILE_SERVER *)
	FS(FSD:=FSD,PT:=R_BUF2); (* Datei von FTP empfangen *)
ELSE
	FS(FSD:=FSD,PT:=S_BUF2); (* Datei an FTP senden *)
END_IF;

(* revision history
ks	11. may 2011	rev 1.2
	ip_control - remote disconnect error ausblenden, und sonderbehandlung für pcworx

ks	06. apr. 2011	rev 1.1
	list_len und list_get durch element_count und element_get ersetzt

ks	01. jan. 2011	rev 1.0
	original version
*)

END_FUNCTION_BLOCK

// oscat_network/POUs/NETWORK/DNS_CLIENT
FUNCTION_BLOCK DNS_CLIENT
VAR_IN_OUT
	IP_C : IP_C; (* IP_Control Verwaltungsstruktur *)
	S_BUF : NETWORK_BUFFER;
	R_BUF : NETWORK_BUFFER;
END_VAR
VAR_INPUT
	ACTIVATE : BOOL;
	DOMAIN : STRING;
	IP4_DNS : DWORD;
END_VAR
VAR_OUTPUT
	IP4 : DWORD;
	DONE : BOOL;
	ERROR : DWORD;
END_VAR
VAR
	IP_FIFO : IP_FIFO;
	ip_state : BYTE;
	ip_id : BYTE;
	i : INT;
	state : INT;
	domain_copy : STRING;
	activate_last : BOOL;
	url_length : INT;
	char : BYTE;
	char_count : INT;
	tid : BYTE;
	anc : INT;
	x : BYTE;
	rr_stop : BOOL;
	ttl_last : DWORD;
	ttl_tmp : DWORD;

	(*LOG_MSG : LOG_MSG;
	_debug_enable : BOOL := TRUE;*)

END_VAR

(*
version 1.3	26. jul. 2011
programmer 	ks
tested BY	ks

DNS_CLIENT führt eine Domain-Name Abfrage bei einen DNS-Server durch

*)

(* Domain Name System (query) *)

CASE state OF

00:	IF ACTIVATE AND NOT activate_last THEN (* auf positive Flanke GET warten *)
		DONE := FALSE;
		ERROR := DWORD#0;
		state := 5;
	END_IF;

05:	IP4 := IP4_DECODE(str:=DOMAIN); (* prüfe ob domain schon eine IP4-Adresse ist *)
	IF IP4 > DWORD#00 THEN
		DONE := TRUE;
		state := 0;
        		(*####################  DEBUG-MESSAGE  ###################################*)
        		(*IF _debug_enable THEN
            		LOG_CL.NEW_MSG := 'DNS: S05 IP4 ~1';
            		LOG_CL.PRINTF[1]  := DOMAIN;
            		LOG_MSG();
        		END_IF;*)
        		(*########################################################################*)
	ELSE
		ip_state := BYTE#1;
		ttl_last := DWORD#0;
		domain_copy := DOMAIN; (* DOMAIN String sichern *)
		state := 10;
        		(*####################  DEBUG-MESSAGE  ###################################*)
        		(*IF _debug_enable THEN
            		LOG_CL.NEW_MSG := 'DNS: S05 START';
            		LOG_MSG();
        		END_IF;*)
        		(*########################################################################*)
	END_IF;

10:	IF ip_state = BYTE#3 THEN (* Bei IP_Control anmelden *)
		url_length := LEN(domain_copy);
		char_count := 17 + url_length; (* sendebuffer initialisieren *)
		FOR i := 0 TO char_count DO
			S_BUF.BUFFER[i] := BYTE#00;
		END_FOR;
		tid := UINT_TO_BYTE(BYTE_TO_UINT(tid) + UINT#1);
		S_BUF.BUFFER[01] := tid; (* Transaction ID lowbyte *)
		S_BUF.BUFFER[02] := BYTE#16#01; (* Flags: highbyte *)
		S_BUF.BUFFER[05] := BYTE#16#01; (* Questions: lowbyte *)
		i := url_length + 12;	(* den servernamen von hinten nach vorne bearbeiten *)
		char_count := 0;
		WHILE i > 12 DO
			char := CODE(STR:=domain_copy,POS:=i - 12);
			IF char = BYTE#46 THEN (* prüfe auf haupt/sub domänen namens-teiler "." *)
				S_BUF.BUFFER[i] := INT_TO_BYTE(char_count); (* anstelle des teilers "." wird die länge des erkannten haupt/sub domänennames eingetragen *)
				char_count := 0;
			ELSE
				S_BUF.BUFFER[i] := char; (* char in buffer eintragen *)
				char_count := char_count + 1; (* anzahl char zählen *)
			END_IF;
			i := i - 1;
		END_WHILE;
		S_BUF.BUFFER[i] := INT_TO_BYTE(char_count); (* längenangabe des ganz linken (ersten) domänennamens eintragen *)
		i := url_length + 15; (* position hinter dem servernamen *)
		S_BUF.BUFFER[i] := BYTE#01; (* Type: A Hostaddress lowbyte *)
		i := i + 2;
		S_BUF.BUFFER[i] := BYTE#01; (* Class: IN lowbyte *)
		i := i + 1;
		(* IP Datenverkehr einrichten *)
		IP_C.C_PORT := WORD#53; (* Portnummer eintragen *)
		IP_C.C_IP := IP4_DNS; (* IP eintragen *)
		IP_C.C_MODE := BYTE#1; (* Mode: UDP+AKTIV+PORT+IP *)
		IP_C.C_ENABLE := TRUE; (* Verbindungsaufbau freigeben *)
		IP_C.TIME_RESET := TRUE; (* Zeitueberwachung rücksetzen *)
		IP_C.R_OBSERVE  := TRUE; (* Datenempfang ueberwachen *)
		S_BUF.SIZE := INT_TO_UINT(i); (* sendelänge eintragen *)
		R_BUF.SIZE := UINT#0; (* Empfangslänge rücksetzen *)
		state := 30;

        		(*####################  DEBUG-MESSAGE  ###################################*)
        		(*IF _debug_enable THEN
            		LOG_CL.NEW_MSG := 'DNS: S10 SEND';
            		LOG_MSG();
        		END_IF;*)
        		(*########################################################################*)
	END_IF;

30:	IF IP_C.ERROR <> DWORD#00 THEN
		ERROR := IP_C.ERROR;
		state := 99;
        		(*####################  DEBUG-MESSAGE  ###################################*)
        		(*IF _debug_enable THEN
            		LOG_CL.NEW_MSG := 'DNS: S30 ERROR ~1';
            		LOG_CL.PRINTF[1]  := DWORD_TO_STRING(ERROR);
            		LOG_MSG();
        		END_IF;*)
        		(*########################################################################*)

	ELSIF (S_BUF.SIZE = UINT#0) AND (tid = R_BUF.BUFFER[1]) AND (R_BUF.SIZE >= INT_TO_UINT(34 + url_length)) THEN	(* prüfe ob antwort telegramm die richtige Transaction-ID und mindestlänge hat *)
		ERROR := BYTE_TO_DWORD(R_BUF.BUFFER[3] AND BYTE#2#0000_1111); (* prüfe Return code der Flags. 4 bits *)
		IF ERROR = DWORD#00 THEN
			anc := R_BUF.BUFFER[7]; (* Anzahl der Answer-RR *)
			IP_C.R_OBSERVE := FALSE; (* Datenempfang ueberwachen *)
			state := 40;
		ELSE
			state := 99;
		END_IF;
	END_IF;

40:	IF anc > 0 THEN
		anc := anc - 1;
		WHILE i < R_BUF.SIZE DO
			x := R_BUF.BUFFER[i];
			IF rr_stop = FALSE THEN
				IF x > BYTE#63 THEN (* zeiger auf namen *)
					i := i + 1;
					rr_stop := TRUE;
				ELSIF x= BYTE#0 THEN (* namens ende *)
					rr_stop := TRUE;
				ELSE
					i := i + x; (* namen *)
				END_IF;
				i := i + 1;
			ELSE
				rr_stop := FALSE;
				IF R_BUF.BUFFER[i+1] = BYTE#1 AND R_BUF.BUFFER[i+3] = BYTE#1 THEN (* Type A / Class IN *)
					i := i + 4;
					ttl_tmp := DWORD_OF_BYTE(R_BUF.BUFFER[i],R_BUF.BUFFER[i+1],R_BUF.BUFFER[i+2],R_BUF.BUFFER[i+3]); (* Time to live *)
					i := i + 6;
					IF ttl_tmp >= ttl_last THEN (* TTL ist länger *)
						ttl_last := ttl_tmp;
						IP4 := DWORD_OF_BYTE(R_BUF.BUFFER[i],R_BUF.BUFFER[i+1],R_BUF.BUFFER[i+2],R_BUF.BUFFER[i+3]); (* IP-Adresse *)
					END_IF;
					i := i + 4;
				ELSE
					i := i + 9;
					i := i + R_BUF.BUFFER[i] + 1; (* offset zu nächsten Block *)
				END_IF;
				EXIT;
			END_IF;
		END_WHILE;
	ELSE
		IF IP4 > DWORD#0 THEN (* gültige RR mit IP gefunden *)
			DONE := TRUE;
            		(*####################  DEBUG-MESSAGE  ###################################*)
            		(*IF _debug_enable THEN
                			LOG_CL.NEW_MSG := 'DNS: S40 OK';
                			LOG_MSG();
            		END_IF;*)
            		(*########################################################################*)
		ELSE
			ERROR := DWORD#255; (* Daten fehlerhaft - keine IP-Adresse vorhanden *)
		END_IF;
		state := 99;
	END_IF;

99:	R_BUF.SIZE := UINT#0; (* Empfangslänge rücksetzen *)
	ip_state := BYTE#4; (* Abmelden *)
	state := 00;

END_CASE;

activate_last := ACTIVATE; (* letzten Status sichern zur Flankenerkennung *)
IP_FIFO(FIFO:=IP_C.FIFO,STATE:=ip_state,ID:=ip_id); (* IP_FIFO *)

(* revision history

ks	18. oct. 2008	rev 1.0
	original version

ks	20. oct. 2009	rev 1.1
	unbenutzten code entfernt, all buffer base 0

ks	20. dec. 2010	rev 1.2
	parsing nach rfc1305

ks	26. jul. 2011	rev 1.3
	verbesserte ip-auswertung , neue fehlermeldung
*)


(*----------------------------------------------------------------------------------------------------------------*)
(* Flags: 0x0100 (Standard query)                                                                                            *)
(* 0... .... .... .... = Response: Message is a query                                                                   *)
(* .000 0... ....  = Opcode: Standard query (0)                                                                          *)
(* .... ..0. .... .... = Truncated: Message is not truncated                                                          *)
(* .... ...1 .... .... = Recursion desired: Do query recursively                                                    *)
(* .... .... .0.. .... = Z: reserved (0)                                                                                                  *)
(* .... .... ...0 .... = Non-authenticated data OK: Non-authenticated data is unacceptable *)
(*-----------------------------------------------------------------------------------------------------------------*)

(*      0  1  2  3  4  5  6  7  8  9  0  1  2  3  4  5  *)
(*    +--+--+--+--+--+--+--+--+--+--+--+--+--+--+--+--+ *)
(*    |                      ID                       | idx: 0/1   *)
(*    +--+--+--+--+--+--+--+--+--+--+--+--+--+--+--+--+ *)
(*    |QR|   Opcode  |AA|TC|RD|RA|   Z    |   RCODE   | idx: 2/3   *)
(*    +--+--+--+--+--+--+--+--+--+--+--+--+--+--+--+--+ *)
(*    |                    QDCOUNT                    | idx: 4/5   *)
(*    +--+--+--+--+--+--+--+--+--+--+--+--+--+--+--+--+ *)
(*    |                    ANCOUNT                    | idx: 6/7   *)
(*    +--+--+--+--+--+--+--+--+--+--+--+--+--+--+--+--+ *)
(*    |                    NSCOUNT                    | idx: 8/9   *)
(*    +--+--+--+--+--+--+--+--+--+--+--+--+--+--+--+--+ *)
(*    |                    ARCOUNT                    | idx: 10/11 *)
(*    +--+--+--+--+--+--+--+--+--+--+--+--+--+--+--+--+ *)

(*
Errorcodes  Description	References 
000	No error. 		 	The request completed successfully.
001	Format error. 		The name server was unable to interpret the query. 
002	Server failure.  	The name server was unable to process this query due to a problem with the name server. 
003	Name Error. 	 	Meaningful only for responses from an authoritative name server, this code signifies that the domain name referenced in the query does not exist.
004	Not Implemented. 	The name server does not support the requested kind of query.
005	Refused. 			The name server refuses to perform the specified operation for policy reasons.
  						 For example, a name server may not wish to provide the information to the particular requester, or a name server may not wish to perform a particular operation (e.g., zone transfer) for particular data.
006	YXDomain.			Name Exists when it should not. 
007	YXRRSet. RR			Set Exists when it should not. 
008	NXRRSet. RR			Set that should exist does not. 
009	NotAuth.			Server Not Authoritative for zone. 
010	NotZone,			Name not contained in zone. 
255	Timeout				No Response  
   

beispiel einer DNS Request von google.at
ein request mit 3 Answer-Blocks


Domain Name System (response)
[Request In: 3]
[Time: 0.027533000 seconds]
Transaction ID: 0x5e1a
Flags: 0x8180 (Standard query response, No error)
1... .... .... .... = Response: Message is a response
.000 0... .... .... = Opcode: Standard query (0)
.... .0.. .... .... = Authoritative: Server is not an authority for domain
.... ..0. .... .... = Truncated: Message is not truncated
.... ...1 .... .... = Recursion desired: Do query recursively
.... .... 1... .... = Recursion available: Server can do recursive queries
.... .... .0.. .... = Z: reserved (0)
.... .... ..0. .... = Answer authenticated: Answer/authority portion was not authenticated
.... .... .... 0000 = Reply code: No error (0)
Questions: 1
Answer RRs: 3
Authority RRs: 0
Additional RRs: 0

Queries
google.at: type A, class IN
Name: google.at
Type: A (Host address)
Class: IN (0x0001)

Answers
google.at: type A, class IN, addr 72.14.221.104
Name: google.at
Type: A (Host address)
Class: IN (0x0001)
Time to live: 19 minutes, 9 seconds
Data length: 4
Addr: 72.14.221.104

google.at: type A, class IN, addr 66.249.93.104
Name: google.at
Type: A (Host address)
Class: IN (0x0001)
Time to live: 19 minutes, 9 seconds
Data length: 4
Addr: 66.249.93.104

google.at: type A, class IN, addr 216.239.59.104
Name: google.at
Type: A (Host address)
Class: IN (0x0001)
Time to live: 19 minutes, 9 seconds
Data length: 4
Addr: 216.239.59.104
*)

END_FUNCTION_BLOCK

// oscat_network/POUs/NETWORK/IP_FIFO
FUNCTION_BLOCK IP_FIFO
VAR_IN_OUT
	FIFO : IP_FIFO_DATA;
	ID : BYTE;
	STATE : BYTE;
END_VAR
VAR
	tmp : INT;

	(*LOG_MSG : LOG_MSG;
	_debug_enable : BOOL := TRUE;*)

END_VAR

(*	version 1.0	18. oct. 2008
	programmer 	ks
	tested BY		ks

	IP_FIFO ist ein Zusatzbaustein füR die Zugriffsverwaltung auf IP_CONTROL
*)

IF NOT FIFO.INIT THEN
	FIFO.INIT := TRUE;
	FIFO.NW := 1;
	FIFO.NR := 1;
	FIFO.EMPTY := TRUE;
	FIFO.FULL := FALSE;
	FIFO.TOP := 128; (* Arraygroesse 1 bis x *)
	FIFO.MAX_ID := BYTE#1; (* maximale anzahl von Anmeldungen einer ID *)
END_IF;

(* wenn keine ID vorhanden dann die naechste freie ID zuteilen *)
IF ID = BYTE#00 THEN
	IF FIFO.ID < INT_TO_BYTE(FIFO.TOP) THEN
		ID := USINT_TO_BYTE(BYTE_TO_USINT(FIFO.ID) + USINT#1); (* ID +1 *)
		FIFO.ID := ID; (* ID eintragen *)
	    	(*####################  DEBUG-MESSAGE  ###################################*)
	    	(*IF _debug_enable THEN
	      		LOG_CL.NEW_MSG := 'FIFO: NEW ID:~1';
	      		LOG_CL.PRINTF[1]  := BYTE_TO_STRING(ID);
	      		LOG_MSG();
	    	END_IF;*)
	    	(*########################################################################*)
	ELSIF STATE < BYTE#200 THEN
		(*####################  DEBUG-MESSAGE  ###################################*)
		(*IF _debug_enable THEN
			LOG_CL.NEW_MSG := 'FIFO: OVERFLOW ADD ID';
			LOG_MSG();
		END_IF;*)
		(*########################################################################*)

		(* sollte nie passieren ! -> es sind zuviele teilnehmer angemeldet *)
		(* es wird keine Nummer vergeben und alle anfragen werden negativ beantwortet *)
		STATE := BYTE#255;
		RETURN;
	END_IF;
END_IF;

